  MoveL 1169 to (549.24, 512.97, 16) mm, rotated rx -180 ry 0 rz 160 deg; joints [7.081, 85.862, -31.558, -147.805, 58.7, 161.888]
  Set speed (17.5 mm/s)
  Call Extruder(1124.88314)
  MoveL 1170 to (548.96, 514.02, 16) mm, rotated rx -180 ry 0 rz 160 deg; joints [7.204, 85.828, -31.485, -147.681, 58.771, 161.841]
  Set speed (17.5 mm/s)
  Call Extruder(1131.34964)
  MoveL 1171 to (548.37, 515.94, 16) mm, rotated rx -180 ry 0 rz 160 deg; joints [7.43, 85.752, -31.322, -147.46, 58.916, 161.767]
  Set speed (17.5 mm/s)
  Call Extruder(1135.34697)
  MoveL 1172 to (547.97, 517.11, 16) mm, rotated rx 180 ry 0 rz 160 deg; joints [7.568, 85.697, -31.202, -147.327, 59.013, 161.728]
  Set speed (17.5 mm/s)
  Call Extruder(1138.01654)
  MoveL 1173 to (547.69, 517.88, 16) mm, rotated rx -180 ry 0 rz 160 deg; joints [7.66, 85.658, -31.119, -147.24, 59.08, 161.704]
  Set speed (17.5 mm/s)
  Call Extruder(1141.53682)
  MoveL 1174 to (547.29, 518.9, 16) mm, rotated rx -180 ry 0 rz 160 deg; joints [7.781, 85.601, -30.995, -147.127, 59.174, 161.677]
  Set speed (17.5 mm/s)
  Call Extruder(1144.91482)
  MoveL 1175 to (546.9, 519.87, 16) mm, rotated rx 180 ry 0 rz 160 deg; joints [7.897, 85.544, -30.872, -147.021, 59.266, 161.653]
  Set speed (17.5 mm/s)
  Call Extruder(1151.46736)
  MoveL 1176 to (546.07, 521.72, 16) mm, rotated rx -180 ry 0 rz 160 deg; joints [8.12, 85.42, -30.605, -146.821, 59.456, 161.619]
  Call Extruder(1154.81875)
  MoveL 1177 to (545.61, 522.65, 16) mm, rotated rx 180 ry 0 rz 160 deg; joints [8.233, 85.352, -30.456, -146.722, 59.559, 161.607]
  Set speed (17.5 mm/s)
  Call Extruder(1158.37572)
  MoveL 1178 to (545.12, 523.64, 16) mm, rotated rx -180 ry 0 rz 160 deg; joints [8.353, 85.275, -30.29, -146.619, 59.671, 161.597]
  Call Extruder(1161.73090)
  MoveL 1179 to (544.62, 524.55, 16) mm, rotated rx 180 ry 0 rz 160 deg; joints [8.465, 85.198, -30.123, -146.525, 59.782, 161.592]
  Set speed (17.5 mm/s)
  Call Extruder(1165.06713)
  MoveL 1180 to (544.12, 525.45, 16) mm, rotated rx -180 ry 0 rz 160 deg; joints [8.576, 85.119, -29.952, -146.433, 59.894, 161.59]
  Set speed (17.5 mm/s)
  Call Extruder(1169.60064)
  MoveL 1181 to (543.4, 526.66, 16) mm, rotated rx 180 ry 0 rz 160 deg; joints [8.726, 85.006, -29.706, -146.311, 60.051, 161.593]
  Set speed (17.5 mm/s)
  Call Extruder(1175.11317)
  MoveL 1182 to (542.48, 528.1, 16) mm, rotated rx 180 ry 0 rz 160 deg; joints [8.905, 84.859, -29.387, -146.17, 60.251, 161.605]
  Set speed (17.5 mm/s)
  Call Extruder(1178.53672)
  MoveL 1183 to (541.88, 528.97, 16) mm, rotated rx -180 ry 0 rz 160 deg; joints [9.016, 84.764, -29.18, -146.085, 60.379, 161.618]
  Set speed (17.5 mm/s)
  Call Extruder(1181.80346)
  MoveL 1184 to (541.3, 529.8, 16) mm, rotated rx 180 ry 0 rz 160 deg; joints [9.12, 84.67, -28.975, -146.005, 60.504, 161.632]
  Call Extruder(1185.22640)
  MoveL 1185 to (540.67, 530.65, 16) mm, rotated rx 180 ry 0 rz 160 deg; joints [9.229, 84.568, -28.753, -145.925, 60.638, 161.651]
  Set speed (17.5 mm/s)
  Call Extruder(1188.52738)
  MoveL 1186 to (540.05, 531.47, 16) mm, rotated rx -180 ry 0 rz 160 deg; joints [9.333, 84.467, -28.534, -145.849, 60.769, 161.672]
  Call Extruder(1191.91987)
  MoveL 1187 to (539.39, 532.28, 16) mm, rotated rx 180 ry 0 rz 160 deg; joints [9.439, 84.361, -28.3, -145.774, 60.907, 161.698]
  Set speed (17.5 mm/s)
  Call Extruder(1195.33158)
  MoveL 1188 to (538.71, 533.09, 16) mm, rotated rx 180 ry 0 rz 160 deg; joints [9.544, 84.25, -28.058, -145.7, 61.049, 161.727]
  Set speed (17.5 mm/s)
  Call Extruder(1198.69325)
  MoveL 1189 to (538.03, 533.88, 16) mm, rotated rx 180 ry 0 rz 160 deg; joints [9.647, 84.139, -27.814, -145.63, 61.19, 161.758]
  Set speed (17.5 mm/s)
  Call Extruder(1202.01515)
  MoveL 1190 to (537.33, 534.64, 16) mm, rotated rx 180 ry 0 rz 160 deg; joints [9.748, 84.026, -27.567, -145.563, 61.333, 161.792]
  Set speed (17.5 mm/s)
  Call Extruder(1205.37905)
  MoveL 1191 to (536.62, 535.4, 16) mm, rotated rx -180 ry 0 rz 160 deg; joints [9.849, 83.909, -27.31, -145.497, 61.479, 161.83]
  Call Extruder(1208.76243)
  MoveL 1192 to (535.88, 536.14, 16) mm, rotated rx -180 ry 0 rz 160 deg; joints [9.949, 83.789, -27.047, -145.432, 61.629, 161.871]
  Call Extruder(1212.12100)
  MoveL 1193 to (535.14, 536.87, 16) mm, rotated rx 180 ry 0 rz 160 deg; joints [10.047, 83.667, -26.779, -145.371, 61.779, 161.915]
  Call Extruder(1215.53799)
  MoveL 1194 to (534.36, 537.59, 16) mm, rotated rx -180 ry 0 rz 160 deg; joints [10.146, 83.541, -26.502, -145.311, 61.934, 161.962]
  Set speed (17.5 mm/s)
  Call Extruder(1218.83854)
  MoveL 1195 to (533.6, 538.27, 16) mm, rotated rx -180 ry 0 rz 160 deg; joints [10.24, 83.417, -26.228, -145.255, 62.087, 162.011]
  Set speed (17.5 mm/s)
  Call Extruder(1222.23079)
  MoveL 1196 to (532.8, 538.96, 16) mm, rotated rx 180 ry 0 rz 160 deg; joints [10.335, 83.287, -25.941, -145.199, 62.245, 162.065]
  Set speed (17.5 mm/s)
  Call Extruder(1225.64774)
  MoveL 1197 to (531.99, 539.63, 16) mm, rotated rx 180 ry 0 rz 160 deg; joints [10.43, 83.154, -25.648, -145.146, 62.406, 162.121]
  Set speed (17.5 mm/s)
  Call Extruder(1228.34274)
  MoveL 1198 to (531.33, 540.15, 16) mm, rotated rx 180 ry 0 rz 160 deg; joints [10.504, 83.048, -25.413, -145.105, 62.534, 162.167]
  Set speed (17.5 mm/s)
  Call Extruder(1232.24907)
  MoveL 1199 to (530.37, 540.88, 16) mm, rotated rx 180 ry 0 rz 160 deg; joints [10.609, 82.892, -25.067, -145.048, 62.722, 162.238]
  Set speed (17.5 mm/s)
  Call Extruder(1235.63039)
  MoveL 1200 to (529.52, 541.5, 16) mm, rotated rx 180 ry 0 rz 160 deg; joints [10.698, 82.755, -24.763, -145.002, 62.886, 162.302]
  Set speed (17.5 mm/s)
  Call Extruder(1238.99206)
  MoveL 1201 to (528.67, 542.1, 16) mm, rotated rx 180 ry 0 rz 160 deg; joints [10.786, 82.617, -24.456, -144.958, 63.051, 162.368]
  Call Extruder(1242.35571)
  MoveL 1202 to (527.8, 542.67, 16) mm, rotated rx -180 ry 0 rz 160 deg; joints [10.872, 82.477, -24.145, -144.916, 63.217, 162.437]
  Set speed (17.5 mm/s)
  Call Extruder(1245.76604)
  MoveL 1203 to (526.91, 543.24, 16) mm, rotated rx -180 ry 0 rz 160 deg; joints [10.958, 82.333, -23.825, -144.875, 63.387, 162.509]
  Set speed (17.5 mm/s)
  Call Extruder(1249.75916)
  MoveL 1204 to (525.85, 543.88, 16) mm, rotated rx 180 ry 0 rz 160 deg; joints [11.056, 82.164, -23.447, -144.83, 63.587, 162.597]
  Set speed (17.5 mm/s)
  Call Extruder(1255.55529)
  MoveL 1205 to (524.29, 544.77, 16) mm, rotated rx 180 ry 0 rz 160 deg; joints [11.195, 81.914, -22.888, -144.771, 63.881, 162.73]
  Set speed (17.5 mm/s)
  Call Extruder(1258.01050)
  MoveL 1206 to (523.62, 545.13, 16) mm, rotated rx -180 ry 0 rz 160 deg; joints [11.252, 81.808, -22.649, -144.747, 64.006, 162.788]
  Set speed (17.5 mm/s)
  Call Extruder(1261.12140)
  MoveL 1207 to (522.76, 545.56, 16) mm, rotated rx 180 ry 0 rz 160 deg; joints [11.323, 81.671, -22.342, -144.719, 64.166, 162.865]
  Set speed (17.5 mm/s)
  Call Extruder(1265.86908)
  MoveL 1208 to (521.44, 546.2, 16) mm, rotated rx 180 ry 0 rz 160 deg; joints [11.428, 81.461, -21.869, -144.681, 64.411, 162.984]
  Set speed (17.5 mm/s)
  Call Extruder(1269.35473)
  MoveL 1209 to (520.45, 546.64, 16) mm, rotated rx 180 ry 0 rz 160 deg; joints [11.503, 81.305, -21.519, -144.655, 64.592, 163.075]
  Call Extruder(1272.87309)
  MoveL 1210 to (519.45, 547.07, 16) mm, rotated rx 180 ry 0 rz 160 deg; joints [11.578, 81.148, -21.164, -144.63, 64.775, 163.168]
  Set speed (17.5 mm/s)
  Call Extruder(1279.51361)
  MoveL 1211 to (517.54, 547.82, 16) mm, rotated rx 180 ry 0 rz 160 deg; joints [11.712, 80.848, -20.484, -144.591, 65.123, 163.351]
  Set speed (17.5 mm/s)
  Call Extruder(1286.22822)
  MoveL 1212 to (515.57, 548.49, 16) mm, rotated rx 180 ry 0 rz 160 deg; joints [11.84, 80.542, -19.789, -144.56, 65.477, 163.543]
  Set speed (17.4 mm/s)
  Call Extruder(1290.32257)
  MoveL 1213 to (514.36, 548.86, 16) mm, rotated rx -180 ry 0 rz 160 deg; joints [11.914, 80.354, -19.361, -144.545, 65.693, 163.663]
  Set speed (17.5 mm/s)
  Call Extruder(1292.76941)
  MoveL 1214 to (513.63, 549.07, 16) mm, rotated rx -180 ry 0 rz 160 deg; joints [11.957, 80.242, -19.105, -144.538, 65.823, 163.736]
  Set speed (17.5 mm/s)
  Call Extruder(1295.71612)
  MoveL 1215 to (512.75, 549.3, 16) mm, rotated rx 180 ry 0 rz 160 deg; joints [12.006, 80.106, -18.794, -144.531, 65.979, 163.826]
  Set speed (17.5 mm/s)
  Call Extruder(1299.58645)
  MoveL 1216 to (511.59, 549.59, 16) mm, rotated rx 180 ry 0 rz 160 deg; joints [12.07, 79.928, -18.386, -144.523, 66.184, 163.945]
  Set speed (17.5 mm/s)
  Call Extruder(1306.36625)
  MoveL 1217 to (509.53, 550.03, 16) mm, rotated rx -180 ry 0 rz 160 deg; joints [12.175, 79.615, -17.666, -144.516, 66.544, 164.159]
  Set speed (17.5 mm/s)
  Call Extruder(1313.14810)
  MoveL 1218 to (507.46, 550.38, 16) mm, rotated rx 180 ry 0 rz 160 deg; joints [12.27, 79.301, -16.941, -144.519, 66.905, 164.379]
  Set speed (17.5 mm/s)
  Call Extruder(1319.69345)
  MoveL 1219 to (505.45, 550.64, 16) mm, rotated rx 180 ry 0 rz 160 deg; joints [12.354, 78.998, -16.239, -144.53, 67.252, 164.596]
  Set speed (17.5 mm/s)
  Call Extruder(1326.55936)
  MoveL 1220 to (503.33, 550.82, 16) mm, rotated rx -180 ry 0 rz 160 deg; joints [12.432, 78.681, -15.501, -144.549, 67.615, 164.829]
  Set speed (17.5 mm/s)
  Call Extruder(1333.32860)
  MoveL 1221 to (501.24, 550.91, 16) mm, rotated rx 180 ry 0 rz 160 deg; joints [12.499, 78.369, -14.774, -144.578, 67.972, 165.063]
  Set speed (17.5 mm/s)
  Call Extruder(1339.97617)
  MoveL 1222 to (499.18, 550.92, 16) mm, rotated rx -180 ry 0 rz 160 deg; joints [12.556, 78.066, -14.061, -144.614, 68.32, 165.297]
  Set speed (10.0 mm/s)
  MoveL 1223 to (499.18, 550.92, 20) mm, rotated rx 180 ry 0 rz 160 deg; joints [12.556, 77.328, -13.499, -144.573, 68.176, 165.187]
  Set speed (120.0 mm/s)
  MoveL 1224 to (499.16, 551.9, 20) mm, rotated rx 180 ry 0 rz 160 deg; joints [12.676, 77.358, -13.57, -144.439, 68.174, 165.115]
  Set speed (17.5 mm/s)
  Call Extruder(1346.89767)
  MoveL 1225 to (497.02, 551.82, 20) mm, rotated rx 180 ry 0 rz 160 deg; joints [12.725, 77.043, -12.831, -144.486, 68.531, 165.362]
  Set speed (17.5 mm/s)
  Call Extruder(1353.77145)
  MoveL 1226 to (494.9, 551.66, 20) mm, rotated rx 180 ry 0 rz 160 deg; joints [12.763, 76.734, -12.101, -144.541, 68.883, 165.609]
  Call Extruder(1360.44876)
  MoveL 1227 to (492.84, 551.41, 20) mm, rotated rx 180 ry 0 rz 160 deg; joints [12.791, 76.436, -11.396, -144.603, 69.222, 165.852]
  Set speed (17.5 mm/s)
  Call Extruder(1367.36675)
  MoveL 1228 to (490.72, 551.07, 20) mm, rotated rx 180 ry 0 rz 160 deg; joints [12.808, 76.131, -10.67, -144.676, 69.57, 166.106]
  Set speed (17.5 mm/s)
  Call Extruder(1374.35141)
  MoveL 1229 to (488.6, 550.64, 20) mm, rotated rx -180 ry 0 rz 160 deg; joints [12.814, 75.828, -9.943, -144.76, 69.917, 166.364]
  Set speed (17.5 mm/s)
  Call Extruder(1381.22915)
  MoveL 1230 to (486.53, 550.13, 20) mm, rotated rx 180 ry 0 rz 160 deg; joints [12.81, 75.533, -9.236, -144.851, 70.253, 166.619]
  Call Extruder(1387.89760)
  MoveL 1231 to (484.55, 549.56, 20) mm, rotated rx 180 ry 0 rz 160 deg; joints [12.794, 75.252, -8.558, -144.948, 70.575, 166.867]
  Set speed (17.5 mm/s)
  Call Extruder(1394.66926)
  MoveL 1232 to (482.56, 548.89, 20) mm, rotated rx 180 ry 0 rz 160 deg; joints [12.767, 74.972, -7.877, -145.057, 70.896, 167.119]
  Set speed (17.5 mm/s)
  Call Extruder(1398.28337)
  MoveL 1233 to (481.51, 548.5, 20) mm, rotated rx 180 ry 0 rz 160 deg; joints [12.747, 74.825, -7.518, -145.118, 71.065, 167.254]
  Call Extruder(1401.87388)
  MoveL 1234 to (480.48, 548.1, 20) mm, rotated rx -180 ry 0 rz 160 deg; joints [12.726, 74.68, -7.164, -145.181, 71.232, 167.387]
  Set speed (17.5 mm/s)
  Call Extruder(1406.78546)
  MoveL 1235 to (479.08, 547.51, 20) mm, rotated rx 180 ry 0 rz 160 deg; joints [12.691, 74.484, -6.685, -145.272, 71.458, 167.569]
  Set speed (17.5 mm/s)
  Call Extruder(1411.85900)
  MoveL 1236 to (477.65, 546.85, 20) mm, rotated rx 180 ry 0 rz 160 deg; joints [12.649, 74.285, -6.196, -145.371, 71.687, 167.757]
  Set speed (17.5 mm/s)
  Call Extruder(1416.96547)
  MoveL 1237 to (476.23, 546.15, 20) mm, rotated rx -180 ry 0 rz 160 deg; joints [12.6, 74.088, -5.71, -145.475, 71.915, 167.945]
  Set speed (17.5 mm/s)
  Call Extruder(1422.63061)
  MoveL 1238 to (474.69, 545.32, 20) mm, rotated rx 180 ry 0 rz 160 deg; joints [12.537, 73.874, -5.18, -145.597, 72.163, 168.153]
  Set speed (17.5 mm/s)
  Call Extruder(1425.60662)
  MoveL 1239 to (473.89, 544.87, 20) mm, rotated rx 180 ry 0 rz 160 deg; joints [12.501, 73.763, -4.905, -145.664, 72.291, 168.262]
  Set speed (17.5 mm/s)
  Call Extruder(1429.03570)
  MoveL 1240 to (472.97, 544.32, 20) mm, rotated rx 180 ry 0 rz 160 deg; joints [12.457, 73.637, -4.591, -145.743, 72.437, 168.387]
  Call Extruder(1432.47238)
  MoveL 1241 to (472.07, 543.76, 20) mm, rotated rx -180 ry 0 rz 160 deg; joints [12.41, 73.513, -4.28, -145.825, 72.582, 168.512]
  Set speed (17.5 mm/s)
  Call Extruder(1435.86869)
  MoveL 1242 to (471.19, 543.18, 20) mm, rotated rx -180 ry 0 rz 160 deg; joints [12.36, 73.391, -3.976, -145.908, 72.723, 168.634]
  Set speed (17.5 mm/s)
  Call Extruder(1439.36515)
  MoveL 1243 to (470.29, 542.57, 20) mm, rotated rx -180 ry 0 rz 160 deg; joints [12.306, 73.268, -3.667, -145.996, 72.867, 168.759]
  Set speed (17.5 mm/s)
  Call Extruder(1442.74341)
  MoveL 1244 to (469.44, 541.96, 20) mm, rotated rx 180 ry 0 rz 160 deg; joints [12.251, 73.151, -3.372, -146.082, 73.003, 168.88]
  Set speed (17.5 mm/s)
  Call Extruder(1446.13527)
  MoveL 1245 to (468.6, 541.34, 20) mm, rotated rx 180 ry 0 rz 160 deg; joints [12.193, 73.035, -3.08, -146.172, 73.139, 169]
  Call Extruder(1449.64837)
  MoveL 1246 to (467.74, 540.67, 20) mm, rotated rx -180 ry 0 rz 160 deg; joints [12.129, 72.917, -2.782, -146.267, 73.276, 169.123]
  Set speed (17.5 mm/s)
  Call Extruder(1453.05307)
  MoveL 1247 to (466.92, 540, 20) mm, rotated rx 180 ry 0 rz 160 deg; joints [12.065, 72.805, -2.497, -146.362, 73.408, 169.242]
  Set speed (17.5 mm/s)
  Call Extruder(1456.40954)
  MoveL 1248 to (466.12, 539.33, 20) mm, rotated rx -180 ry 0 rz 160 deg; joints [11.999, 72.696, -2.22, -146.457, 73.536, 169.358]
  Set speed (17.5 mm/s)
  Call Extruder(1459.89153)
  MoveL 1249 to (465.31, 538.62, 20) mm, rotated rx 180 ry 0 rz 160 deg; joints [11.927, 72.585, -1.937, -146.558, 73.666, 169.478]
  Call Extruder(1463.26727)
  MoveL 1250 to (464.54, 537.91, 20) mm, rotated rx 180 ry 0 rz 160 deg; joints [11.855, 72.479, -1.667, -146.659, 73.79, 169.593]
  Set speed (17.5 mm/s)
  Call Extruder(1466.74547)
  MoveL 1251 to (463.76, 537.17, 20) mm, rotated rx -180 ry 0 rz 160 deg; joints [11.778, 72.372, -1.393, -146.764, 73.916, 169.71]
  Set speed (17.5 mm/s)
  Call Extruder(1470.14894)
  MoveL 1252 to (463.01, 536.42, 20) mm, rotated rx 180 ry 0 rz 160 deg; joints [11.7, 72.27, -1.13, -146.869, 74.036, 169.824]
  Set speed (17.5 mm/s)
  Call Extruder(1473.62936)
  MoveL 1253 to (462.26, 535.64, 20) mm, rotated rx -180 ry 0 rz 160 deg; joints [11.617, 72.167, -0.866, -146.98, 74.157, 169.939]
  Set speed (17.5 mm/s)
  Call Extruder(1476.95452)
  MoveL 1254 to (461.56, 534.89, 20) mm, rotated rx 180 ry 0 rz 160 deg; joints [11.535, 72.071, -0.618, -147.087, 74.27, 170.047]
  Set speed (17.5 mm/s)
  Call Extruder(1480.45766)
  MoveL 1255 to (460.84, 534.08, 20) mm, rotated rx -180 ry 0 rz 160 deg; joints [11.446, 71.972, -0.362, -147.202, 74.387, 170.161]
  Set speed (17.5 mm/s)
  Call Extruder(1483.42207)
  MoveL 1256 to (460.24, 533.38, 20) mm, rotated rx 180 ry 0 rz 160 deg; joints [11.368, 71.89, -0.149, -147.301, 74.483, 170.255]
  Set speed (17.5 mm/s)
  Call Extruder(1487.30579)
  MoveL 1257 to (459.48, 532.45, 20) mm, rotated rx 180 ry 0 rz 160 deg; joints [11.264, 71.785, 0.124, -147.433, 74.607, 170.378]
  Set speed (17.5 mm/s)
  Call Extruder(1490.73127)
  MoveL 1258 to (458.83, 531.62, 20) mm, rotated rx -180 ry 0 rz 160 deg; joints [11.168, 71.694, 0.359, -147.552, 74.713, 170.484]
  Set speed (17.5 mm/s)
  Call Extruder(1494.14375)
  MoveL 1259 to (458.19, 530.77, 20) mm, rotated rx -180 ry 0 rz 160 deg; joints [11.071, 71.606, 0.588, -147.672, 74.816, 170.589]
  Set speed (17.5 mm/s)
  Call Extruder(1497.58334)
  MoveL 1260 to (457.57, 529.9, 20) mm, rotated rx -180 ry 0 rz 160 deg; joints [10.97, 71.52, 0.814, -147.795, 74.918, 170.693]
  Set speed (17.5 mm/s)
  Call Extruder(1500.98572)
  MoveL 1261 to (456.97, 529.04, 20) mm, rotated rx 180 ry 0 rz 160 deg; joints [10.867, 71.437, 1.032, -147.919, 75.016, 170.794]
  Set speed (17.5 mm/s)
  Call Extruder(1504.45910)
  MoveL 1262 to (456.38, 528.14, 20) mm, rotated rx 180 ry 0 rz 160 deg; joints [10.761, 71.354, 1.25, -148.048, 75.113, 170.896]
  Set speed (17.5 mm/s)
  Call Extruder(1507.83348)
  MoveL 1263 to (455.82, 527.25, 20) mm, rotated rx -180 ry 0 rz 160 deg; joints [10.654, 71.276, 1.455, -148.174, 75.204, 170.994]
  Set speed (17.5 mm/s)
  Call Extruder(1511.23944)
  MoveL 1264 to (455.27, 526.35, 20) mm, rotated rx 180 ry 0 rz 160 deg; joints [10.545, 71.199, 1.657, -148.303, 75.294, 171.09]
  Call Extruder(1514.69572)
  MoveL 1265 to (454.74, 525.42, 20) mm, rotated rx -180 ry 0 rz 160 deg; joints [10.431, 71.124, 1.857, -148.436, 75.382, 171.187]
  Set speed (17.5 mm/s)
  Call Extruder(1517.51539)
  MoveL 1266 to (454.32, 524.66, 20) mm, rotated rx 180 ry 0 rz 160 deg; joints [10.337, 71.064, 2.015, -148.546, 75.451, 171.264]
  Set speed (17.5 mm/s)
  Call Extruder(1521.55599)
  MoveL 1267 to (453.74, 523.55, 20) mm, rotated rx 180 ry 0 rz 160 deg; joints [10.199, 70.981, 2.234, -148.706, 75.547, 171.373]
  Set speed (17.5 mm/s)
  Call Extruder(1524.99033)
  MoveL 1268 to (453.26, 522.59, 20) mm, rotated rx 180 ry 0 rz 160 deg; joints [10.079, 70.913, 2.415, -148.843, 75.626, 171.464]
  Set speed (17.5 mm/s)
  Call Extruder(1528.51455)
  MoveL 1269 to (452.8, 521.61, 20) mm, rotated rx 180 ry 0 rz 160 deg; joints [9.954, 70.846, 2.593, -148.985, 75.702, 171.555]
  Set speed (17.5 mm/s)
  Call Extruder(1531.83917)
  MoveL 1270 to (452.38, 520.67, 20) mm, rotated rx -180 ry 0 rz 160 deg; joints [9.834, 70.785, 2.757, -149.121, 75.773, 171.639]
  Set speed (17.5 mm/s)
  Call Extruder(1538.58210)
  MoveL 1271 to (451.59, 518.73, 20) mm, rotated rx -180 ry 0 rz 160 deg; joints [9.585, 70.668, 3.07, -149.401, 75.905, 171.805]
  Call Extruder(1545.63097)
  MoveL 1272 to (450.84, 516.68, 20) mm, rotated rx -180 ry 0 rz 160 deg; joints [9.316, 70.555, 3.373, -149.699, 76.031, 171.971]
  Call Extruder(1552.49327)
  MoveL 1273 to (450.2, 514.66, 20) mm, rotated rx 180 ry 0 rz 160 deg; joints [9.048, 70.455, 3.642, -149.994, 76.14, 172.124]
  Set speed (17.5 mm/s)
  Call Extruder(1559.18400)
  MoveL 1274 to (449.65, 512.65, 20) mm, rotated rx -180 ry 0 rz 160 deg; joints [8.779, 70.367, 3.88, -150.286, 76.234, 172.266]
  Set speed (17.5 mm/s)
  Call Extruder(1562.76659)
  MoveL 1275 to (449.4, 511.57, 20) mm, rotated rx 180 ry 0 rz 160 deg; joints [8.633, 70.324, 3.996, -150.443, 76.278, 172.339]
  Call Extruder(1566.05852)
  MoveL 1276 to (449.18, 510.58, 20) mm, rotated rx 180 ry 0 rz 160 deg; joints [8.498, 70.286, 4.098, -150.589, 76.316, 172.404]
  Set speed (17.5 mm/s)
  Call Extruder(1573.08116)
  MoveL 1277 to (448.78, 508.44, 20) mm, rotated rx -180 ry 0 rz 160 deg; joints [8.205, 70.214, 4.295, -150.903, 76.386, 172.537]
  Call Extruder(0.00000)
  Set speed (17.5 mm/s)
  Call Extruder(6.84930)
  MoveL 1278 to (448.48, 506.34, 20) mm, rotated rx -180 ry 0 rz 160 deg; joints [7.914, 70.153, 4.46, -151.212, 76.44, 172.659]
  Set speed (17.5 mm/s)
  Call Extruder(13.69641)
  MoveL 1279 to (448.26, 504.23, 20) mm, rotated rx 180 ry 0 rz 160 deg; joints [7.62, 70.102, 4.599, -151.522, 76.48, 172.772]
  Set speed (17.5 mm/s)
  Call Extruder(20.39008)
  MoveL 1280 to (448.13, 502.16, 20) mm, rotated rx -180 ry 0 rz 160 deg; joints [7.329, 70.062, 4.709, -151.827, 76.505, 172.876]
  Call Extruder(27.31483)
  MoveL 1281 to (448.09, 500.02, 20) mm, rotated rx 180 ry 0 rz 160 deg; joints [7.026, 70.03, 4.795, -152.143, 76.516, 172.974]
  Set speed (17.5 mm/s)
  Call Extruder(33.56591)
  MoveL 1282 to (448.13, 498.08, 20) mm, rotated rx 180 ry 0 rz 160 deg; joints [6.75, 70.01, 4.85, -152.428, 76.513, 173.056]
  Set speed (17.5 mm/s)
  Call Extruder(39.66263)
  MoveL 1283 to (448.23, 496.19, 20) mm, rotated rx -180 ry 0 rz 160 deg; joints [6.48, 69.998, 4.881, -152.706, 76.498, 173.13]
  Call Extruder(46.07765)
  MoveL 1284 to (448.41, 494.21, 20) mm, rotated rx 180 ry 0 rz 160 deg; joints [6.195, 69.995, 4.891, -152.997, 76.47, 173.201]
  Set speed (17.5 mm/s)
  Call Extruder(51.90887)
  MoveL 1285 to (448.65, 492.42, 20) mm, rotated rx 180 ry 0 rz 160 deg; joints [5.936, 69.999, 4.879, -153.261, 76.432, 173.26]
  Call Extruder(58.24782)
  MoveL 1286 to (448.97, 490.48, 20) mm, rotated rx -180 ry 0 rz 160 deg; joints [5.656, 70.012, 4.845, -153.545, 76.38, 173.317]
  Set speed (17.5 mm/s)
  Call Extruder(64.31632)
  MoveL 1287 to (449.35, 488.64, 20) mm, rotated rx 180 ry 0 rz 160 deg; joints [5.388, 70.032, 4.79, -153.815, 76.318, 173.366]
  Set speed (17.5 mm/s)
  Call Extruder(70.48045)
  MoveL 1288 to (449.8, 486.78, 20) mm, rotated rx -180 ry 0 rz 160 deg; joints [5.118, 70.06, 4.712, -154.086, 76.242, 173.409]
  Set speed (17.5 mm/s)
  Call Extruder(76.66227)
  MoveL 1289 to (450.32, 484.94, 20) mm, rotated rx 180 ry 0 rz 160 deg; joints [4.849, 70.097, 4.612, -154.354, 76.155, 173.446]
  Set speed (17.5 mm/s)
  Call Extruder(82.76319)
  MoveL 1290 to (450.9, 483.14, 20) mm, rotated rx -180 ry 0 rz 160 deg; joints [4.586, 70.141, 4.492, -154.615, 76.056, 173.477]
  Call Extruder(89.07136)
  MoveL 1291 to (451.57, 481.31, 20) mm, rotated rx -180 ry 0 rz 160 deg; joints [4.317, 70.195, 4.346, -154.881, 75.942, 173.503]
  Call Extruder(95.23992)
  MoveL 1292 to (452.29, 479.54, 20) mm, rotated rx -180 ry 0 rz 160 deg; joints [4.058, 70.255, 4.182, -155.135, 75.819, 173.523]
  Call Extruder(101.24751)
  MoveL 1293 to (453.06, 477.84, 20) mm, rotated rx 180 ry 0 rz 160 deg; joints [3.81, 70.322, 4.001, -155.377, 75.687, 173.536]
  Set speed (17.5 mm/s)
  Call Extruder(107.57777)
  MoveL 1294 to (453.93, 476.08, 20) mm, rotated rx -180 ry 0 rz 160 deg; joints [3.553, 70.4, 3.79, -155.627, 75.537, 173.544]
  Call Extruder(113.65141)
  MoveL 1295 to (454.83, 474.43, 20) mm, rotated rx 180 ry 0 rz 160 deg; joints [3.312, 70.483, 3.567, -155.86, 75.382, 173.547]
  Set speed (17.5 mm/s)
  Call Extruder(119.90561)
  MoveL 1296 to (455.81, 472.76, 20) mm, rotated rx 180 ry 0 rz 160 deg; joints [3.068, 70.576, 3.315, -156.093, 75.21, 173.544]
  Set speed (17.5 mm/s)
  Call Extruder(125.99893)
  MoveL 1297 to (456.83, 471.17, 20) mm, rotated rx -180 ry 0 rz 160 deg; joints [2.837, 70.675, 3.051, -156.313, 75.033, 173.536]
  Set speed (17.5 mm/s)
  Call Extruder(132.15800)
  MoveL 1298 to (457.92, 469.6, 20) mm, rotated rx -180 ry 0 rz 160 deg; joints [2.609, 70.782, 2.764, -156.528, 74.843, 173.522]
  Call Extruder(138.31119)
  MoveL 1299 to (459.07, 468.07, 20) mm, rotated rx 180 ry 0 rz 160 deg; joints [2.388, 70.897, 2.458, -156.735, 74.642, 173.504]
  Set speed (17.5 mm/s)
  Call Extruder(144.56702)
  MoveL 1300 to (460.29, 466.57, 20) mm, rotated rx 180 ry 0 rz 160 deg; joints [2.171, 71.022, 2.127, -156.937, 74.428, 173.479]
  Set speed (17.5 mm/s)
  Call Extruder(150.65295)
  MoveL 1301 to (461.53, 465.15, 20) mm, rotated rx -180 ry 0 rz 160 deg; joints [1.966, 71.15, 1.787, -157.124, 74.209, 173.45]
  Set speed (17.5 mm/s)
  Call Extruder(156.90741)
  MoveL 1302 to (462.86, 463.74, 20) mm, rotated rx 180 ry 0 rz 160 deg; joints [1.764, 71.29, 1.418, -157.308, 73.975, 173.416]
  Call Extruder(162.86927)
  MoveL 1303 to (464.17, 462.44, 20) mm, rotated rx -180 ry 0 rz 160 deg; joints [1.579, 71.43, 1.05, -157.475, 73.743, 173.378]
  Call Extruder(169.18566)
  MoveL 1304 to (465.61, 461.11, 20) mm, rotated rx 180 ry 0 rz 160 deg; joints [1.39, 71.586, 0.642, -157.641, 73.488, 173.332]
  Set speed (17.5 mm/s)
  Call Extruder(175.35316)
  MoveL 1305 to (467.07, 459.87, 20) mm, rotated rx 180 ry 0 rz 160 deg; joints [1.215, 71.745, 0.226, -157.794, 73.231, 173.283]
  Set speed (17.5 mm/s)
  Call Extruder(181.85609)
  MoveL 1306 to (468.65, 458.63, 20) mm, rotated rx -180 ry 0 rz 160 deg; joints [1.039, 71.921, -0.23, -157.944, 72.95, 173.225]
  Set speed (17.5 mm/s)
  Call Extruder(187.18333)
  MoveL 1307 to (469.98, 457.65, 20) mm, rotated rx 180 ry 0 rz 160 deg; joints [0.903, 72.071, -0.617, -158.058, 72.714, 173.174]
  Set speed (17.5 mm/s)
  Call Extruder(193.82493)
  MoveL 1308 to (471.68, 456.49, 20) mm, rotated rx -180 ry 0 rz 160 deg; joints [0.742, 72.264, -1.116, -158.19, 72.412, 173.105]
  Set speed (17.5 mm/s)
  Call Extruder(200.07187)
  MoveL 1309 to (473.32, 455.47, 20) mm, rotated rx 180 ry 0 rz 160 deg; joints [0.6, 72.454, -1.602, -158.303, 72.119, 173.035]
  Call Extruder(206.24160)
  MoveL 1310 to (474.98, 454.52, 20) mm, rotated rx -180 ry 0 rz 160 deg; joints [0.469, 72.648, -2.097, -158.403, 71.824, 172.96]
  Set speed (17.5 mm/s)
  Call Extruder(212.42019)
  MoveL 1311 to (476.67, 453.63, 20) mm, rotated rx 180 ry 0 rz 160 deg; joints [0.348, 72.848, -2.606, -158.493, 71.521, 172.881]
  Set speed (17.5 mm/s)
  Call Extruder(218.39493)
  MoveL 1312 to (478.34, 452.83, 20) mm, rotated rx -180 ry 0 rz 160 deg; joints [0.239, 73.048, -3.112, -158.569, 71.223, 172.799]
  Call Extruder(224.75574)
  MoveL 1313 to (480.15, 452.04, 20) mm, rotated rx 180 ry 0 rz 160 deg; joints [0.133, 73.267, -3.664, -158.639, 70.9, 172.707]
  Set speed (17.5 mm/s)
  Call Extruder(230.75775)
  MoveL 1314 to (481.88, 451.36, 20) mm, rotated rx 180 ry 0 rz 160 deg; joints [0.041, 73.48, -4.197, -158.694, 70.59, 172.615]
  Set speed (17.5 mm/s)
  Call Extruder(237.09101)
  MoveL 1315 to (483.73, 450.71, 20) mm, rotated rx 180 ry 0 rz 160 deg; joints [-0.045, 73.71, -4.771, -158.74, 70.258, 172.513]
  Set speed (17.5 mm/s)
  Call Extruder(243.20984)
  MoveL 1316 to (485.54, 450.14, 20) mm, rotated rx 180 ry 0 rz 160 deg; joints [-0.118, 73.937, -5.337, -158.773, 69.933, 172.409]
  Set speed (17.5 mm/s)
  Call Extruder(249.37088)
  MoveL 1317 to (487.39, 449.65, 20) mm, rotated rx -180 ry 0 rz 160 deg; joints [-0.183, 74.172, -5.918, -158.796, 69.602, 172.299]
  Call Extruder(255.54669)
  MoveL 1318 to (489.25, 449.21, 20) mm, rotated rx -180 ry 0 rz 160 deg; joints [-0.239, 74.413, -6.51, -158.807, 69.266, 172.184]
  Set speed (17.5 mm/s)
  Call Extruder(261.60188)
  MoveL 1319 to (491.09, 448.86, 20) mm, rotated rx 180 ry 0 rz 160 deg; joints [-0.284, 74.653, -7.1, -158.807, 68.934, 172.066]
  Set speed (17.5 mm/s)
  Call Extruder(267.49098)
  MoveL 1320 to (492.89, 448.58, 20) mm, rotated rx -180 ry 0 rz 160 deg; joints [-0.32, 74.891, -7.681, -158.796, 68.609, 171.946]
  Call Extruder(273.99527)
  MoveL 1321 to (494.9, 448.34, 20) mm, rotated rx -180 ry 0 rz 160 deg; joints [-0.348, 75.159, -8.332, -158.772, 68.248, 171.808]
  Set speed (17.5 mm/s)
  Call Extruder(280.16768)
  MoveL 1322 to (496.8, 448.19, 20) mm, rotated rx -180 ry 0 rz 160 deg; joints [-0.367, 75.418, -8.957, -158.738, 67.904, 171.672]
  Call Extruder(286.42584)
  MoveL 1323 to (498.74, 448.11, 20) mm, rotated rx 180 ry 0 rz 160 deg; joints [-0.376, 75.684, -9.598, -158.692, 67.553, 171.529]
  Set speed (17.5 mm/s)
  Call Extruder(292.51904)
  MoveL 1324 to (500.63, 448.09, 20) mm, rotated rx 180 ry 0 rz 160 deg; joints [-0.376, 75.947, -10.229, -158.636, 67.211, 171.384]
  Set speed (17.5 mm/s)
  Call Extruder(298.76296)
  MoveL 1325 to (502.56, 448.15, 20) mm, rotated rx -180 ry 0 rz 160 deg; joints [-0.367, 76.219, -10.88, -158.568, 66.859, 171.23]
  Set speed (17.5 mm/s)
  Call Extruder(304.84597)
  MoveL 1326 to (504.44, 448.28, 20) mm, rotated rx -180 ry 0 rz 160 deg; joints [-0.349, 76.488, -11.52, -158.49, 66.517, 171.075]
  Set speed (17.5 mm/s)
  Call Extruder(310.88075)
  MoveL 1327 to (506.3, 448.48, 20) mm, rotated rx -180 ry 0 rz 160 deg; joints [-0.323, 76.758, -12.158, -158.403, 66.179, 170.916]
  Set speed (17.5 mm/s)
  Call Extruder(317.20333)
  MoveL 1328 to (508.24, 448.75, 20) mm, rotated rx -180 ry 0 rz 160 deg; joints [-0.287, 77.042, -12.829, -158.301, 65.825, 170.744]
  Set speed (17.5 mm/s)
  Call Extruder(323.33518)
  MoveL 1329 to (510.11, 449.08, 20) mm, rotated rx 180 ry 0 rz 160 deg; joints [-0.244, 77.321, -13.483, -158.192, 65.483, 170.572]
  Set speed (17.5 mm/s)
  Call Extruder(328.91158)
  MoveL 1330 to (511.8, 449.45, 20) mm, rotated rx 180 ry 0 rz 160 deg; joints [-0.198, 77.575, -14.079, -158.083, 65.174, 170.412]
  Call Extruder(335.60217)
  MoveL 1331 to (513.81, 449.96, 20) mm, rotated rx 180 ry 0 rz 160 deg; joints [-0.134, 77.882, -14.794, -157.942, 64.806, 170.213]
  Set speed (17.5 mm/s)
  Call Extruder(341.84087)
  MoveL 1332 to (515.67, 450.51, 20) mm, rotated rx 180 ry 0 rz 160 deg; joints [-0.066, 78.17, -15.462, -157.8, 64.466, 170.023]
  Set speed (17.5 mm/s)
  Call Extruder(348.08429)
  MoveL 1333 to (517.5, 451.13, 20) mm, rotated rx -180 ry 0 rz 160 deg; joints [0.011, 78.459, -16.129, -157.647, 64.129, 169.827]
  Call Extruder(354.17423)
  MoveL 1334 to (519.27, 451.8, 20) mm, rotated rx -180 ry 0 rz 160 deg; joints [0.092, 78.741, -16.779, -157.489, 63.803, 169.632]
  Call Extruder(360.41686)
  MoveL 1335 to (521.05, 452.55, 20) mm, rotated rx -180 ry 0 rz 160 deg; joints [0.183, 79.03, -17.443, -157.318, 63.474, 169.427]
  Call Extruder(366.58690)
  MoveL 1336 to (522.78, 453.36, 20) mm, rotated rx -180 ry 0 rz 160 deg; joints [0.281, 79.315, -18.095, -157.139, 63.153, 169.22]
  Set speed (17.5 mm/s)
  Call Extruder(372.59726)
  MoveL 1337 to (524.44, 454.21, 20) mm, rotated rx 180 ry 0 rz 160 deg; joints [0.382, 79.592, -18.726, -156.957, 62.847, 169.014]
  Call Extruder(378.91663)
  MoveL 1338 to (526.15, 455.16, 20) mm, rotated rx -180 ry 0 rz 160 deg; joints [0.496, 79.882, -19.385, -156.757, 62.529, 168.793]
  Set speed (17.5 mm/s)
  Call Extruder(384.99300)
  MoveL 1339 to (527.76, 456.14, 20) mm, rotated rx -180 ry 0 rz 160 deg; joints [0.612, 80.159, -20.013, -156.556, 62.23, 168.577]
  Set speed (17.5 mm/s)
  Call Extruder(391.25117)
  MoveL 1340 to (529.38, 457.21, 20) mm, rotated rx 180 ry 0 rz 160 deg; joints [0.738, 80.442, -20.652, -156.341, 61.929, 168.351]
  Set speed (17.5 mm/s)
  Call Extruder(397.19940)
  MoveL 1341 to (530.88, 458.27, 20) mm, rotated rx 180 ry 0 rz 160 deg; joints [0.863, 80.709, -21.252, -156.13, 61.649, 168.133]
  Set speed (17.5 mm/s)
  Call Extruder(403.53259)
  MoveL 1342 to (532.44, 459.47, 20) mm, rotated rx -180 ry 0 rz 160 deg; joints [1.003, 80.99, -21.882, -155.897, 61.36, 167.897]
  Call Extruder(409.53413)
  MoveL 1343 to (533.87, 460.66, 20) mm, rotated rx -180 ry 0 rz 160 deg; joints [1.14, 81.253, -22.469, -155.67, 61.092, 167.671]
  Call Extruder(415.76527)
  MoveL 1344 to (535.31, 461.95, 20) mm, rotated rx -180 ry 0 rz 160 deg; joints [1.289, 81.521, -23.068, -155.428, 60.824, 167.434]
  Call Extruder(422.07973)
  MoveL 1345 to (536.72, 463.3, 20) mm, rotated rx -180 ry 0 rz 160 deg; joints [1.445, 81.789, -23.664, -155.177, 60.56, 167.191]
  Call Extruder(425.35628)
  MoveL 1346 to (537.43, 464.03, 20) mm, rotated rx 180 ry 0 rz 160 deg; joints [1.528, 81.926, -23.968, -155.044, 60.428, 167.065]
  Set speed (17.5 mm/s)
  Call Extruder(428.77503)
  MoveL 1347 to (538.15, 464.8, 20) mm, rotated rx 180 ry 0 rz 160 deg; joints [1.617, 82.067, -24.28, -154.903, 60.292, 166.932]
  Set speed (17.5 mm/s)
  Call Extruder(432.19134)
  MoveL 1348 to (538.86, 465.59, 20) mm, rotated rx -180 ry 0 rz 160 deg; joints [1.707, 82.206, -24.589, -154.761, 60.159, 166.799]
  Set speed (17.5 mm/s)
  Call Extruder(435.63311)
  MoveL 1349 to (539.56, 466.39, 20) mm, rotated rx -180 ry 0 rz 160 deg; joints [1.799, 82.345, -24.895, -154.617, 60.029, 166.665]
  Set speed (17.5 mm/s)
  Call Extruder(439.17845)
  MoveL 1350 to (540.27, 467.24, 20) mm, rotated rx -180 ry 0 rz 160 deg; joints [1.895, 82.486, -25.205, -154.467, 59.898, 166.527]
  Set speed (17.5 mm/s)
  Call Extruder(442.52401)
  MoveL 1351 to (540.91, 468.05, 20) mm, rotated rx -180 ry 0 rz 160 deg; joints [1.987, 82.617, -25.494, -154.323, 59.777, 166.396]
  Set speed (17.5 mm/s)
  Call Extruder(445.90952)
  MoveL 1352 to (541.55, 468.88, 20) mm, rotated rx -180 ry 0 rz 160 deg; joints [2.082, 82.747, -25.781, -154.177, 59.659, 166.264]
  Set speed (17.5 mm/s)
  Call Extruder(448.86173)
  MoveL 1353 to (542.09, 469.62, 20) mm, rotated rx 180 ry 0 rz 160 deg; joints [2.165, 82.859, -26.028, -154.049, 59.557, 166.148]
  Call Extruder(452.72753)
  MoveL 1354 to (542.78, 470.6, 20) mm, rotated rx 180 ry 0 rz 160 deg; joints [2.276, 83.003, -26.343, -153.88, 59.43, 165.997]
  Set speed (17.5 mm/s)
  Call Extruder(455.75332)
  MoveL 1355 to (543.31, 471.38, 20) mm, rotated rx -180 ry 0 rz 160 deg; joints [2.364, 83.114, -26.587, -153.746, 59.332, 165.879]
  Call Extruder(459.59881)
  MoveL 1356 to (543.95, 472.38, 20) mm, rotated rx -180 ry 0 rz 160 deg; joints [2.477, 83.252, -26.889, -153.575, 59.213, 165.729]
  Set speed (17.5 mm/s)
  Call Extruder(463.01746)
  MoveL 1357 to (544.51, 473.28, 20) mm, rotated rx -180 ry 0 rz 160 deg; joints [2.579, 83.372, -27.151, -153.422, 59.111, 165.596]
  Set speed (17.5 mm/s)
  Call Extruder(466.46723)
  MoveL 1358 to (545.05, 474.21, 20) mm, rotated rx 180 ry 0 rz 160 deg; joints [2.683, 83.49, -27.41, -153.267, 59.011, 165.462]
  Set speed (17.5 mm/s)
  Call Extruder(471.90101)
  MoveL 1359 to (545.86, 475.68, 20) mm, rotated rx -180 ry 0 rz 160 deg; joints [2.848, 83.671, -27.805, -153.022, 58.862, 165.253]
  Set speed (17.5 mm/s)
  Call Extruder(476.86174)
  MoveL 1360 to (546.56, 477.05, 20) mm, rotated rx -180 ry 0 rz 160 deg; joints [3.002, 83.83, -28.15, -152.797, 58.735, 165.063]
  Set speed (17.5 mm/s)
  Call Extruder(482.73409)
  MoveL 1361 to (547.34, 478.69, 20) mm, rotated rx -180 ry 0 rz 160 deg; joints [3.186, 84.011, -28.545, -152.529, 58.594, 164.84]
  Set speed (17.5 mm/s)
  Call Extruder(490.40334)
  MoveL 1362 to (548.26, 480.88, 20) mm, rotated rx 180 ry 0 rz 160 deg; joints [3.432, 84.231, -29.022, -152.178, 58.43, 164.555]
  Set speed (17.5 mm/s)
  Call Extruder(497.19049)
  MoveL 1363 to (548.99, 482.85, 20) mm, rotated rx -180 ry 0 rz 160 deg; joints [3.653, 84.413, -29.416, -151.867, 58.303, 164.307]
  Set speed (17.5 mm/s)
  Call Extruder(500.81084)
  MoveL 1364 to (549.35, 483.91, 20) mm, rotated rx 180 ry 0 rz 160 deg; joints [3.772, 84.503, -29.612, -151.701, 58.242, 164.178]
  Set speed (17.5 mm/s)
  Call Extruder(504.13273)
  MoveL 1365 to (549.66, 484.89, 20) mm, rotated rx 180 ry 0 rz 160 deg; joints [3.881, 84.585, -29.789, -151.549, 58.188, 164.059]
  Set speed (17.5 mm/s)
  Call Extruder(511.08636)
  MoveL 1366 to (550.25, 486.97, 20) mm, rotated rx 180 ry 0 rz 160 deg; joints [4.113, 84.743, -30.13, -151.232, 58.091, 163.817]
  Call Extruder(517.86034)
  MoveL 1367 to (550.73, 489.01, 20) mm, rotated rx 180 ry 0 rz 160 deg; joints [4.342, 84.881, -30.429, -150.925, 58.015, 163.589]
  Call Extruder(524.78335)
  MoveL 1368 to (551.14, 491.11, 20) mm, rotated rx 180 ry 0 rz 160 deg; joints [4.578, 85.008, -30.701, -150.614, 57.955, 163.364]
  Call Extruder(531.56213)
  MoveL 1369 to (551.46, 493.19, 20) mm, rotated rx -180 ry 0 rz 160 deg; joints [4.811, 85.115, -30.932, -150.312, 57.914, 163.152]
  Set speed (17.5 mm/s)
  Call Extruder(538.57711)
  MoveL 1370 to (551.7, 495.35, 20) mm, rotated rx 180 ry 0 rz 160 deg; joints [5.054, 85.21, -31.137, -150.003, 57.89, 162.942]
  Set speed (17.5 mm/s)
  Call Extruder(545.33174)
  MoveL 1371 to (551.85, 497.44, 20) mm, rotated rx 180 ry 0 rz 160 deg; joints [5.29, 85.285, -31.297, -149.711, 57.886, 162.75]
  Set speed (17.5 mm/s)
  Call Extruder(552.17049)
  MoveL 1372 to (551.91, 499.56, 20) mm, rotated rx -180 ry 0 rz 160 deg; joints [5.529, 85.343, -31.423, -149.419, 57.899, 162.566]
  Set speed (17.5 mm/s)
  Call Extruder(559.11146)
  MoveL 1373 to (551.88, 501.71, 20) mm, rotated rx 180 ry 0 rz 160 deg; joints [5.773, 85.385, -31.513, -149.13, 57.931, 162.391]
  Set speed (17.5 mm/s)
  Call Extruder(565.86897)
  MoveL 1374 to (551.77, 503.8, 20) mm, rotated rx 180 ry 0 rz 160 deg; joints [6.011, 85.408, -31.562, -148.854, 57.981, 162.233]
  Call Extruder(572.64602)
  MoveL 1375 to (551.57, 505.89, 20) mm, rotated rx -180 ry 0 rz 160 deg; joints [6.25, 85.415, -31.576, -148.583, 58.048, 162.087]
  Set speed (17.5 mm/s)
  Call Extruder(579.67802)
  MoveL 1376 to (551.28, 508.05, 20) mm, rotated rx -180 ry 0 rz 160 deg; joints [6.498, 85.403, -31.551, -148.31, 58.136, 161.948]
  Set speed (17.5 mm/s)
  Call Extruder(586.42842)
  MoveL 1377 to (550.92, 510.11, 20) mm, rotated rx 180 ry 0 rz 160 deg; joints [6.735, 85.375, -31.49, -148.055, 58.237, 161.828]
  Set speed (17.5 mm/s)
  Call Extruder(593.33712)
  MoveL 1378 to (550.46, 512.21, 20) mm, rotated rx 180 ry 0 rz 160 deg; joints [6.978, 85.328, -31.39, -147.801, 58.358, 161.719]
  Set speed (17.5 mm/s)
  Call Extruder(596.73152)
  MoveL 1379 to (550.19, 513.22, 20) mm, rotated rx 180 ry 0 rz 160 deg; joints [7.096, 85.298, -31.325, -147.681, 58.425, 161.672]
  Set speed (17.5 mm/s)
  Call Extruder(600.32140)
  MoveL 1380 to (549.9, 514.3, 20) mm, rotated rx -180 ry 0 rz 160 deg; joints [7.222, 85.263, -31.251, -147.554, 58.498, 161.624]
  Set speed (17.5 mm/s)
  Call Extruder(606.81202)
  MoveL 1381 to (549.31, 516.22, 20) mm, rotated rx 180 ry 0 rz 160 deg; joints [7.448, 85.187, -31.086, -147.332, 58.644, 161.548]
  Call Extruder(613.77511)
  MoveL 1382 to (548.6, 518.26, 20) mm, rotated rx 180 ry 0 rz 160 deg; joints [7.689, 85.089, -30.876, -147.102, 58.815, 161.481]
  Set speed (17.5 mm/s)
  Call Extruder(620.57631)
  MoveL 1383 to (547.81, 520.21, 20) mm, rotated rx 180 ry 0 rz 160 deg; joints [7.922, 84.976, -30.633, -146.886, 58.998, 161.43]
  Set speed (17.5 mm/s)
  Call Extruder(624.13088)
  MoveL 1384 to (547.37, 521.22, 20) mm, rotated rx -180 ry 0 rz 160 deg; joints [8.043, 84.91, -30.491, -146.777, 59.1, 161.41]
  Set speed (17.5 mm/s)
  Call Extruder(627.38632)
  MoveL 1385 to (546.95, 522.14, 20) mm, rotated rx -180 ry 0 rz 160 deg; joints [8.153, 84.848, -30.357, -146.679, 59.196, 161.394]
  Set speed (17.5 mm/s)
  Call Extruder(630.88513)
  MoveL 1386 to (546.48, 523.11, 20) mm, rotated rx 180 ry 0 rz 160 deg; joints [8.271, 84.776, -30.202, -146.576, 59.303, 161.38]
  Set speed (17.5 mm/s)
  Call Extruder(634.33475)
  MoveL 1387 to (546, 524.07, 20) mm, rotated rx -180 ry 0 rz 160 deg; joints [8.387, 84.702, -30.042, -146.476, 59.412, 161.37]
  Set speed (17.5 mm/s)
  Call Extruder(637.83411)
  MoveL 1388 to (545.48, 525.02, 20) mm, rotated rx -180 ry 0 rz 160 deg; joints [8.504, 84.622, -29.87, -146.378, 59.526, 161.364]
  Set speed (17.5 mm/s)
  Call Extruder(641.18121)
  MoveL 1389 to (544.97, 525.93, 20) mm, rotated rx -180 ry 0 rz 160 deg; joints [8.615, 84.543, -29.697, -146.286, 59.639, 161.362]
  Set speed (17.5 mm/s)
  Call Extruder(645.47650)
  MoveL 1390 to (544.29, 527.07, 20) mm, rotated rx 180 ry 0 rz 160 deg; joints [8.757, 84.436, -29.466, -146.171, 59.787, 161.364]
  Set speed (17.5 mm/s)
  Call Extruder(648.04286)
  MoveL 1391 to (543.87, 527.75, 20) mm, rotated rx 180 ry 0 rz 160 deg; joints [8.841, 84.369, -29.32, -146.104, 59.879, 161.368]
  Set speed (17.5 mm/s)
  Call Extruder(651.48165)
  MoveL 1392 to (543.29, 528.64, 20) mm, rotated rx -180 ry 0 rz 160 deg; joints [8.953, 84.276, -29.12, -146.017, 60.004, 161.376]
  Set speed (17.5 mm/s)
  Call Extruder(654.87230)
  MoveL 1393 to (542.71, 529.51, 20) mm, rotated rx -180 ry 0 rz 160 deg; joints [9.062, 84.182, -28.916, -145.933, 60.13, 161.388]
  Call Extruder(658.36623)
  MoveL 1394 to (542.08, 530.4, 20) mm, rotated rx 180 ry 0 rz 160 deg; joints [9.174, 84.081, -28.697, -145.848, 60.264, 161.403]
  Set speed (17.5 mm/s)
  Call Extruder(661.88724)
  MoveL 1395 to (541.43, 531.27, 20) mm, rotated rx 180 ry 0 rz 160 deg; joints [9.286, 83.977, -28.47, -145.766, 60.401, 161.422]
  Set speed (17.5 mm/s)
  Call Extruder(665.17030)
  MoveL 1396 to (540.81, 532.08, 20) mm, rotated rx 180 ry 0 rz 160 deg; joints [9.389, 83.877, -28.252, -145.691, 60.531, 161.443]
  Set speed (17.5 mm/s)
  Call Extruder(668.59493)
  MoveL 1397 to (540.15, 532.91, 20) mm, rotated rx 180 ry 0 rz 160 deg; joints [9.496, 83.769, -28.017, -145.615, 60.67, 161.468]
  Set speed (17.5 mm/s)
  Call Extruder(672.08025)
  MoveL 1398 to (539.45, 533.74, 20) mm, rotated rx -180 ry 0 rz 160 deg; joints [9.604, 83.656, -27.771, -145.54, 60.814, 161.497]
  Set speed (17.5 mm/s)
  Call Extruder(675.49297)
  MoveL 1399 to (538.76, 534.53, 20) mm, rotated rx -180 ry 0 rz 160 deg; joints [9.708, 83.543, -27.525, -145.469, 60.957, 161.528]
  Call Extruder(678.85590)
  MoveL 1400 to (538.06, 535.3, 20) mm, rotated rx -180 ry 0 rz 160 deg; joints [9.81, 83.429, -27.275, -145.401, 61.101, 161.563]
  Set speed (17.5 mm/s)
  Call Extruder(682.37940)
  MoveL 1401 to (537.31, 536.1, 20) mm, rotated rx 180 ry 0 rz 160 deg; joints [9.915, 83.306, -27.008, -145.332, 61.253, 161.602]
  Set speed (17.5 mm/s)
  Call Extruder(685.79723)
  MoveL 1402 to (536.56, 536.85, 20) mm, rotated rx -180 ry 0 rz 160 deg; joints [10.016, 83.185, -26.742, -145.268, 61.404, 161.643]
  Set speed (17.5 mm/s)
  Call Extruder(689.14305)
  MoveL 1403 to (535.82, 537.57, 20) mm, rotated rx -180 ry 0 rz 160 deg; joints [10.114, 83.063, -26.476, -145.207, 61.553, 161.686]
  Set speed (17.5 mm/s)
  Call Extruder(695.21264)
  MoveL 1404 to (534.43, 538.85, 20) mm, rotated rx 180 ry 0 rz 160 deg; joints [10.288, 82.838, -25.982, -145.101, 61.829, 161.772]
  Set speed (17.5 mm/s)
  Call Extruder(699.40855)
  MoveL 1405 to (533.45, 539.7, 20) mm, rotated rx -180 ry 0 rz 160 deg; joints [10.406, 82.678, -25.63, -145.033, 62.023, 161.837]
  Set speed (17.5 mm/s)
  Call Extruder(702.90545)
  MoveL 1406 to (532.62, 540.39, 20) mm, rotated rx -180 ry 0 rz 160 deg; joints [10.503, 82.542, -25.331, -144.978, 62.187, 161.894]
  Set speed (17.5 mm/s)
  Call Extruder(706.26813)
  MoveL 1407 to (531.8, 541.03, 20) mm, rotated rx -180 ry 0 rz 160 deg; joints [10.595, 82.41, -25.039, -144.928, 62.346, 161.951]
  Set speed (17.5 mm/s)
  Call Extruder(709.70068)
  MoveL 1408 to (530.95, 541.67, 20) mm, rotated rx -180 ry 0 rz 160 deg; joints [10.688, 82.273, -24.735, -144.879, 62.511, 162.013]
  Set speed (17.5 mm/s)
  Call Extruder(713.15736)
  MoveL 1409 to (530.08, 542.31, 20) mm, rotated rx -180 ry 0 rz 160 deg; joints [10.779, 82.133, -24.426, -144.831, 62.677, 162.078]
  Set speed (17.5 mm/s)
  Call Extruder(716.56707)
  MoveL 1410 to (529.22, 542.91, 20) mm, rotated rx 180 ry 0 rz 160 deg; joints [10.868, 81.992, -24.115, -144.787, 62.844, 162.145]
  Set speed (17.5 mm/s)
  Call Extruder(720.01045)
  MoveL 1411 to (528.33, 543.5, 20) mm, rotated rx 180 ry 0 rz 160 deg; joints [10.956, 81.849, -23.798, -144.744, 63.013, 162.215]
  Set speed (17.5 mm/s)
  Call Extruder(723.39249)
  MoveL 1412 to (527.44, 544.06, 20) mm, rotated rx -180 ry 0 rz 160 deg; joints [11.041, 81.707, -23.482, -144.704, 63.181, 162.286]
  Set speed (17.5 mm/s)
  Call Extruder(726.96845)
  MoveL 1413 to (526.5, 544.64, 20) mm, rotated rx -180 ry 0 rz 160 deg; joints [11.13, 81.556, -23.145, -144.663, 63.359, 162.364]
  Set speed (17.5 mm/s)
  Call Extruder(730.28187)
  MoveL 1414 to (525.61, 545.16, 20) mm, rotated rx -180 ry 0 rz 160 deg; joints [11.21, 81.413, -22.828, -144.629, 63.526, 162.439]
  Set speed (17.5 mm/s)
  Call Extruder(733.10921)
  MoveL 1415 to (524.84, 545.58, 20) mm, rotated rx -180 ry 0 rz 160 deg; joints [11.277, 81.292, -22.556, -144.6, 63.668, 162.504]
  Set speed (17.5 mm/s)
  Call Extruder(739.07113)
  MoveL 1416 to (523.21, 546.44, 20) mm, rotated rx 180 ry 0 rz 160 deg; joints [11.414, 81.032, -21.975, -144.546, 63.971, 162.647]
  Set speed (17.5 mm/s)
  Call Extruder(743.92927)
  MoveL 1417 to (521.85, 547.09, 20) mm, rotated rx 180 ry 0 rz 160 deg; joints [11.522, 80.817, -21.494, -144.506, 64.22, 162.769]
  Call Extruder(747.49721)
  MoveL 1418 to (520.85, 547.54, 20) mm, rotated rx -180 ry 0 rz 160 deg; joints [11.599, 80.658, -21.137, -144.48, 64.404, 162.861]
  Set speed (17.5 mm/s)
  Call Extruder(750.90332)
  MoveL 1419 to (519.88, 547.96, 20) mm, rotated rx 180 ry 0 rz 160 deg; joints [11.671, 80.506, -20.795, -144.456, 64.58, 162.95]
  Set speed (17.5 mm/s)
  Call Extruder(757.79659)
  MoveL 1420 to (517.89, 548.73, 20) mm, rotated rx 180 ry 0 rz 160 deg; joints [11.811, 80.194, -20.092, -144.416, 64.939, 163.139]
  Set speed (17.5 mm/s)
  Call Extruder(764.48818)
  MoveL 1421 to (515.93, 549.41, 20) mm, rotated rx 180 ry 0 rz 160 deg; joints [11.939, 79.889, -19.402, -144.385, 65.289, 163.33]
  Set speed (17.5 mm/s)
  Call Extruder(768.04357)
  MoveL 1422 to (514.88, 549.73, 20) mm, rotated rx 180 ry 0 rz 160 deg; joints [12.003, 79.726, -19.032, -144.372, 65.476, 163.434]
  Set speed (17.5 mm/s)
  Call Extruder(771.49078)
  MoveL 1423 to (513.85, 550.03, 20) mm, rotated rx 180 ry 0 rz 160 deg; joints [12.065, 79.568, -18.673, -144.361, 65.657, 163.536]
  Set speed (17.5 mm/s)
  Call Extruder(774.36838)
  MoveL 1424 to (512.99, 550.26, 20) mm, rotated rx 180 ry 0 rz 160 deg; joints [12.113, 79.436, -18.37, -144.354, 65.808, 163.623]
  Set speed (17.5 mm/s)
  Call Extruder(778.29441)
  MoveL 1425 to (511.81, 550.55, 20) mm, rotated rx -180 ry 0 rz 160 deg; joints [12.178, 79.255, -17.958, -144.346, 66.015, 163.743]
  Set speed (17.5 mm/s)
  Call Extruder(785.18925)
  MoveL 1426 to (509.72, 550.99, 20) mm, rotated rx -180 ry 0 rz 160 deg; joints [12.285, 78.936, -17.228, -144.34, 66.379, 163.96]
  Set speed (17.5 mm/s)
  Call Extruder(792.11012)
  MoveL 1427 to (507.61, 551.35, 20) mm, rotated rx 180 ry 0 rz 160 deg; joints [12.383, 78.616, -16.491, -144.343, 66.744, 164.184]
  Set speed (17.5 mm/s)
  Call Extruder(798.87602)
  MoveL 1428 to (505.53, 551.62, 20) mm, rotated rx 180 ry 0 rz 160 deg; joints [12.469, 78.303, -15.769, -144.353, 67.1, 164.407]
  Set speed (17.5 mm/s)
  Call Extruder(805.77220)
  MoveL 1429 to (503.4, 551.8, 20) mm, rotated rx 180 ry 0 rz 160 deg; joints [12.548, 77.985, -15.032, -144.373, 67.462, 164.64]
  Set speed (17.5 mm/s)
  Call Extruder(812.67959)
  MoveL 1430 to (501.26, 551.9, 20) mm, rotated rx -180 ry 0 rz 160 deg; joints [12.618, 77.667, -14.292, -144.402, 67.823, 164.878]
  Set speed (17.5 mm/s)
  Call Extruder(819.43681)
  MoveL 1431 to (499.16, 551.9, 20) mm, rotated rx 180 ry 0 rz 160 deg; joints [12.676, 77.358, -13.57, -144.439, 68.174, 165.115]
  Set speed (10.0 mm/s)
  MoveL 1432 to (499.16, 551.9, 24) mm, rotated rx -180 ry 0 rz 160 deg; joints [12.676, 76.625, -13.023, -144.395, 68.023, 164.999]
  Set speed (120.0 mm/s)
  MoveL 1433 to (499.17, 552.87, 24) mm, rotated rx 180 ry 0 rz 160 deg; joints [12.793, 76.659, -13.102, -144.262, 68.017, 164.925]
  Set speed (17.5 mm/s)
  Call Extruder(826.56048)
  MoveL 1434 to (496.97, 552.79, 24) mm, rotated rx 180 ry 0 rz 160 deg; joints [12.845, 76.335, -12.344, -144.31, 68.382, 165.177]
  Call Extruder(833.57135)
  MoveL 1435 to (494.8, 552.62, 24) mm, rotated rx -180 ry 0 rz 160 deg; joints [12.885, 76.019, -11.602, -144.366, 68.738, 165.429]
  Set speed (17.5 mm/s)
  Call Extruder(840.47728)
  MoveL 1436 to (492.67, 552.37, 24) mm, rotated rx -180 ry 0 rz 160 deg; joints [12.913, 75.711, -10.876, -144.43, 69.086, 165.679]
  Set speed (17.5 mm/s)
  Call Extruder(847.34597)
  MoveL 1437 to (490.57, 552.03, 24) mm, rotated rx -180 ry 0 rz 160 deg; joints [12.931, 75.408, -10.158, -144.503, 69.428, 165.931]
  Set speed (17.5 mm/s)
  Call Extruder(854.52226)
  MoveL 1438 to (488.39, 551.59, 24) mm, rotated rx 180 ry 0 rz 160 deg; joints [12.938, 75.096, -9.414, -144.589, 69.781, 166.195]
  Set speed (17.5 mm/s)
  Call Extruder(857.92060)
  MoveL 1439 to (487.37, 551.35, 24) mm, rotated rx 180 ry 0 rz 160 deg; joints [12.937, 74.95, -9.065, -144.633, 69.946, 166.321]
  Set speed (17.5 mm/s)
  Call Extruder(861.29157)
  MoveL 1440 to (486.35, 551.09, 24) mm, rotated rx 180 ry 0 rz 160 deg; joints [12.934, 74.806, -8.72, -144.679, 70.109, 166.445]
  Set speed (17.5 mm/s)
  Call Extruder(863.41682)
  MoveL 1441 to (485.72, 550.91, 24) mm, rotated rx -180 ry 0 rz 160 deg; joints [12.931, 74.716, -8.504, -144.708, 70.211, 166.524]
  Set speed (17.5 mm/s)
  Call Extruder(868.53685)
  MoveL 1442 to (484.2, 550.47, 24) mm, rotated rx 180 ry 0 rz 160 deg; joints [12.918, 74.5, -7.986, -144.784, 70.455, 166.714]
  Set speed (17.5 mm/s)
  Call Extruder(875.33211)
  MoveL 1443 to (482.2, 549.8, 24) mm, rotated rx -180 ry 0 rz 160 deg; joints [12.891, 74.219, -7.306, -144.892, 70.775, 166.967]
  Set speed (17.5 mm/s)
  Call Extruder(882.17346)
  MoveL 1444 to (480.22, 549.04, 24) mm, rotated rx 180 ry 0 rz 160 deg; joints [12.853, 73.94, -6.63, -145.01, 71.092, 167.221]
  Set speed (17.5 mm/s)
  Call Extruder(885.86718)
  MoveL 1445 to (479.16, 548.6, 24) mm, rotated rx 180 ry 0 rz 160 deg; joints [12.827, 73.792, -6.27, -145.078, 71.261, 167.358]
  Set speed (17.5 mm/s)
  Call Extruder(889.19058)
  MoveL 1446 to (478.22, 548.19, 24) mm, rotated rx 180 ry 0 rz 160 deg; joints [12.802, 73.661, -5.948, -145.141, 71.411, 167.481]
  Set speed (17.5 mm/s)
  Call Extruder(892.96922)
  MoveL 1447 to (477.16, 547.69, 24) mm, rotated rx -180 ry 0 rz 160 deg; joints [12.77, 73.513, -5.585, -145.215, 71.58, 167.621]
  Set speed (17.5 mm/s)
  Call Extruder(898.02989)
  MoveL 1448 to (475.75, 547, 24) mm, rotated rx -180 ry 0 rz 160 deg; joints [12.722, 73.317, -5.106, -145.319, 71.803, 167.807]
  Call Extruder(903.78619)
  MoveL 1449 to (474.18, 546.15, 24) mm, rotated rx 180 ry 0 rz 160 deg; joints [12.658, 73.099, -4.569, -145.443, 72.053, 168.018]
  Set speed (17.5 mm/s)
  Call Extruder(906.67486)
  MoveL 1450 to (473.41, 545.71, 24) mm, rotated rx 180 ry 0 rz 160 deg; joints [12.624, 72.992, -4.302, -145.507, 72.177, 168.123]
  Set speed (17.5 mm/s)
  Call Extruder(910.22332)
  MoveL 1451 to (472.46, 545.14, 24) mm, rotated rx -180 ry 0 rz 160 deg; joints [12.578, 72.861, -3.978, -145.589, 72.327, 168.253]
  Set speed (17.5 mm/s)
  Call Extruder(913.65325)
  MoveL 1452 to (471.56, 544.58, 24) mm, rotated rx 180 ry 0 rz 160 deg; joints [12.531, 72.736, -3.668, -145.671, 72.47, 168.377]
  Set speed (17.5 mm/s)
  Call Extruder(917.25863)
  MoveL 1453 to (470.62, 543.97, 24) mm, rotated rx 180 ry 0 rz 160 deg; joints [12.479, 72.607, -3.346, -145.759, 72.619, 168.507]
  Set speed (17.5 mm/s)
  Call Extruder(920.60623)
  MoveL 1454 to (469.76, 543.38, 24) mm, rotated rx 180 ry 0 rz 160 deg; joints [12.427, 72.489, -3.051, -145.843, 72.755, 168.627]
  Set speed (17.5 mm/s)
  Call Extruder(924.13307)
  MoveL 1455 to (468.87, 542.75, 24) mm, rotated rx 180 ry 0 rz 160 deg; joints [12.37, 72.366, -2.744, -145.934, 72.896, 168.752]
  Set speed (17.5 mm/s)
  Call Extruder(927.75971)
  MoveL 1456 to (467.97, 542.08, 24) mm, rotated rx 180 ry 0 rz 160 deg; joints [12.308, 72.242, -2.432, -146.029, 73.04, 168.881]
  Set speed (17.5 mm/s)
  Call Extruder(931.15008)
  MoveL 1457 to (467.14, 541.43, 24) mm, rotated rx 180 ry 0 rz 160 deg; joints [12.247, 72.128, -2.145, -146.121, 73.172, 169]
  Set speed (17.5 mm/s)
  Call Extruder(934.63562)
  MoveL 1458 to (466.3, 540.75, 24) mm, rotated rx 180 ry 0 rz 160 deg; joints [12.181, 72.013, -1.855, -146.218, 73.305, 169.121]
  Set speed (17.5 mm/s)
  Call Extruder(938.21784)
  MoveL 1459 to (465.45, 540.04, 24) mm, rotated rx -180 ry 0 rz 160 deg; joints [12.111, 71.896, -1.559, -146.32, 73.44, 169.245]
  Set speed (17.5 mm/s)
  Call Extruder(941.57813)
  MoveL 1460 to (464.67, 539.35, 24) mm, rotated rx 180 ry 0 rz 160 deg; joints [12.042, 71.788, -1.287, -146.417, 73.565, 169.36]
  Set speed (17.5 mm/s)
  Call Extruder(945.08837)
  MoveL 1461 to (463.87, 538.61, 24) mm, rotated rx -180 ry 0 rz 160 deg; joints [11.967, 71.678, -1.007, -146.522, 73.692, 169.48]
  Set speed (17.5 mm/s)
  Call Extruder(948.56346)
  MoveL 1462 to (463.09, 537.87, 24) mm, rotated rx 180 ry 0 rz 160 deg; joints [11.89, 71.571, -0.735, -146.627, 73.816, 169.597]
  Call Extruder(952.05589)
  MoveL 1463 to (462.32, 537.1, 24) mm, rotated rx 180 ry 0 rz 160 deg; joints [11.81, 71.466, -0.465, -146.735, 73.939, 169.713]
  Set speed (17.5 mm/s)
  Call Extruder(955.52014)
  MoveL 1464 to (461.57, 536.33, 24) mm, rotated rx 180 ry 0 rz 160 deg; joints [11.727, 71.363, -0.203, -146.845, 74.058, 169.828]
  Call Extruder(959.04805)
  MoveL 1465 to (460.83, 535.53, 24) mm, rotated rx 180 ry 0 rz 160 deg; joints [11.64, 71.261, 0.059, -146.958, 74.177, 169.943]
  Set speed (17.5 mm/s)
  Call Extruder(962.48274)
  MoveL 1466 to (460.12, 534.73, 24) mm, rotated rx 180 ry 0 rz 160 deg; joints [11.553, 71.163, 0.31, -147.071, 74.29, 170.054]
  Set speed (17.5 mm/s)
  Call Extruder(966.03960)
  MoveL 1467 to (459.41, 533.89, 24) mm, rotated rx -180 ry 0 rz 160 deg; joints [11.46, 71.065, 0.565, -147.19, 74.405, 170.167]
  Call Extruder(969.50471)
  MoveL 1468 to (458.73, 533.06, 24) mm, rotated rx 180 ry 0 rz 160 deg; joints [11.366, 70.971, 0.807, -147.309, 74.514, 170.277]
  Set speed (17.5 mm/s)
  Call Extruder(975.04286)
  MoveL 1469 to (457.67, 531.71, 24) mm, rotated rx 180 ry 0 rz 160 deg; joints [11.211, 70.825, 1.185, -147.501, 74.684, 170.448]
  Set speed (17.5 mm/s)
  Call Extruder(979.97316)
  MoveL 1470 to (456.78, 530.47, 24) mm, rotated rx -180 ry 0 rz 160 deg; joints [11.067, 70.7, 1.509, -147.678, 74.828, 170.598]
  Set speed (17.5 mm/s)
  Call Extruder(983.49957)
  MoveL 1471 to (456.16, 529.57, 24) mm, rotated rx 180 ry 0 rz 160 deg; joints [10.961, 70.614, 1.734, -147.806, 74.928, 170.703]
  Set speed (17.5 mm/s)
  Call Extruder(986.97520)
  MoveL 1472 to (455.57, 528.67, 24) mm, rotated rx 180 ry 0 rz 160 deg; joints [10.854, 70.531, 1.951, -147.935, 75.024, 170.805]
  Call Extruder(990.43757)
  MoveL 1473 to (454.99, 527.76, 24) mm, rotated rx 180 ry 0 rz 160 deg; joints [10.745, 70.451, 2.161, -148.065, 75.117, 170.905]
  Set speed (17.5 mm/s)
  Call Extruder(993.94483)
  MoveL 1474 to (454.43, 526.83, 24) mm, rotated rx -180 ry 0 rz 160 deg; joints [10.632, 70.372, 2.369, -148.198, 75.208, 171.004]
  Set speed (17.5 mm/s)
  Call Extruder(999.57610)
  MoveL 1475 to (453.56, 525.31, 24) mm, rotated rx 180 ry 0 rz 160 deg; joints [10.445, 70.249, 2.692, -148.416, 75.35, 171.162]
  Set speed (17.5 mm/s)
  Call Extruder(1004.34335)
  MoveL 1476 to (452.88, 524, 24) mm, rotated rx 180 ry 0 rz 160 deg; joints [10.282, 70.151, 2.951, -148.605, 75.462, 171.29]
  Set speed (17.5 mm/s)
  Call Extruder(1007.81098)
  MoveL 1477 to (452.4, 523.03, 24) mm, rotated rx -180 ry 0 rz 160 deg; joints [10.161, 70.082, 3.133, -148.744, 75.541, 171.382]
  Set speed (17.5 mm/s)
  Call Extruder(1011.43849)
  MoveL 1478 to (451.93, 522.02, 24) mm, rotated rx -180 ry 0 rz 160 deg; joints [10.032, 70.013, 3.316, -148.891, 75.619, 171.476]
  Call Extruder(1015.01560)
  MoveL 1479 to (451.47, 521.01, 24) mm, rotated rx 180 ry 0 rz 160 deg; joints [9.903, 69.946, 3.492, -149.037, 75.694, 171.567]
  Set speed (17.5 mm/s)
  Call Extruder(1021.92576)
  MoveL 1480 to (450.66, 519.02, 24) mm, rotated rx -180 ry 0 rz 160 deg; joints [9.647, 69.826, 3.812, -149.324, 75.828, 171.737]
  Set speed (17.5 mm/s)
  Call Extruder(1028.73801)
  MoveL 1481 to (449.94, 517.04, 24) mm, rotated rx 180 ry 0 rz 160 deg; joints [9.387, 69.717, 4.104, -149.613, 75.948, 171.897]
  Set speed (17.5 mm/s)
  Call Extruder(1032.49116)
  MoveL 1482 to (449.58, 515.93, 24) mm, rotated rx -180 ry 0 rz 160 deg; joints [9.24, 69.661, 4.253, -149.774, 76.008, 171.982]
  Set speed (17.5 mm/s)
  Call Extruder(1035.74077)
  MoveL 1483 to (449.28, 514.97, 24) mm, rotated rx 180 ry 0 rz 160 deg; joints [9.112, 69.614, 4.378, -149.915, 76.058, 172.054]
  Set speed (17.5 mm/s)
  Call Extruder(1042.69747)
  MoveL 1484 to (448.72, 512.89, 24) mm, rotated rx -180 ry 0 rz 160 deg; joints [8.833, 69.522, 4.625, -150.219, 76.154, 172.202]
  Set speed (17.5 mm/s)
  Call Extruder(1045.73635)
  MoveL 1485 to (448.5, 511.97, 24) mm, rotated rx 180 ry 0 rz 160 deg; joints [8.709, 69.485, 4.724, -150.353, 76.192, 172.264]
  Set speed (17.5 mm/s)
  Call Extruder(1049.60496)
  MoveL 1486 to (448.24, 510.8, 24) mm, rotated rx -180 ry 0 rz 160 deg; joints [8.55, 69.44, 4.845, -150.525, 76.236, 172.341]
  Set speed (17.5 mm/s)
  Call Extruder(1056.82533)
  MoveL 1487 to (447.82, 508.6, 24) mm, rotated rx 180 ry 0 rz 160 deg; joints [8.248, 69.366, 5.047, -150.848, 76.307, 172.479]
  Set speed (17.5 mm/s)
  Call Extruder(1063.81841)
  MoveL 1488 to (447.52, 506.46, 24) mm, rotated rx 180 ry 0 rz 160 deg; joints [7.95, 69.303, 5.215, -151.164, 76.362, 172.603]
  Set speed (17.5 mm/s)
  Call Extruder(1070.79812)
  MoveL 1489 to (447.3, 504.3, 24) mm, rotated rx 180 ry 0 rz 160 deg; joints [7.649, 69.251, 5.357, -151.482, 76.401, 172.72]
  Set speed (17.5 mm/s)
  Call Extruder(1077.59235)
  MoveL 1490 to (447.16, 502.2, 24) mm, rotated rx -180 ry 0 rz 160 deg; joints [7.353, 69.21, 5.468, -151.792, 76.426, 172.825]
  Set speed (17.5 mm/s)
  Call Extruder(1084.65688)
  MoveL 1491 to (447.12, 500.01, 24) mm, rotated rx 180 ry 0 rz 160 deg; joints [7.042, 69.177, 5.556, -152.115, 76.437, 172.926]
  Set speed (17.5 mm/s)
  Call Extruder(1091.01512)
  MoveL 1492 to (447.15, 498.04, 24) mm, rotated rx 180 ry 0 rz 160 deg; joints [6.761, 69.157, 5.612, -152.406, 76.433, 173.01]
  Call Extruder(1097.14303)
  MoveL 1493 to (447.26, 496.14, 24) mm, rotated rx -180 ry 0 rz 160 deg; joints [6.489, 69.145, 5.643, -152.687, 76.418, 173.085]
  Set speed (17.5 mm/s)
  Call Extruder(1103.49292)
  MoveL 1494 to (447.44, 494.19, 24) mm, rotated rx 180 ry 0 rz 160 deg; joints [6.206, 69.142, 5.654, -152.976, 76.39, 173.156]
  Set speed (17.5 mm/s)
  Call Extruder(1109.77189)
  MoveL 1495 to (447.69, 492.25, 24) mm, rotated rx -180 ry 0 rz 160 deg; joints [5.927, 69.146, 5.641, -153.261, 76.35, 173.22]
  Set speed (17.5 mm/s)
  Call Extruder(1115.88410)
  MoveL 1496 to (448, 490.38, 24) mm, rotated rx 180 ry 0 rz 160 deg; joints [5.655, 69.158, 5.608, -153.536, 76.299, 173.276]
  Set speed (17.5 mm/s)
  Call Extruder(1122.26414)
  MoveL 1497 to (448.4, 488.44, 24) mm, rotated rx -180 ry 0 rz 160 deg; joints [5.373, 69.179, 5.551, -153.821, 76.234, 173.328]
  Set speed (17.5 mm/s)
  Call Extruder(1128.63884)
  MoveL 1498 to (448.87, 486.52, 24) mm, rotated rx 180 ry 0 rz 160 deg; joints [5.092, 69.209, 5.47, -154.102, 76.156, 173.373]
  Set speed (17.5 mm/s)
  Call Extruder(1134.87677)
  MoveL 1499 to (449.39, 484.66, 24) mm, rotated rx -180 ry 0 rz 160 deg; joints [4.82, 69.246, 5.37, -154.374, 76.067, 173.412]
  Call Extruder(1141.09003)
  MoveL 1500 to (449.99, 482.83, 24) mm, rotated rx 180 ry 0 rz 160 deg; joints [4.551, 69.291, 5.248, -154.641, 75.967, 173.444]
  Set speed (17.5 mm/s)
  Call Extruder(1147.50044)
  MoveL 1501 to (450.67, 480.96, 24) mm, rotated rx -180 ry 0 rz 160 deg; joints [4.278, 69.346, 5.1, -154.911, 75.851, 173.471]
  Set speed (17.5 mm/s)
  Call Extruder(1153.79361)
  MoveL 1502 to (451.4, 479.15, 24) mm, rotated rx 180 ry 0 rz 160 deg; joints [4.013, 69.408, 4.932, -155.171, 75.726, 173.492]
  Set speed (17.5 mm/s)
  Call Extruder(1160.07652)
  MoveL 1503 to (452.2, 477.37, 24) mm, rotated rx -180 ry 0 rz 160 deg; joints [3.752, 69.478, 4.744, -155.426, 75.589, 173.507]
  Set speed (17.5 mm/s)
  Call Extruder(1166.21648)
  MoveL 1504 to (453.05, 475.67, 24) mm, rotated rx 180 ry 0 rz 160 deg; joints [3.503, 69.554, 4.539, -155.668, 75.443, 173.516]
  Call Extruder(1172.53589)
  MoveL 1505 to (453.98, 473.95, 24) mm, rotated rx 180 ry 0 rz 160 deg; joints [3.251, 69.641, 4.307, -155.911, 75.282, 173.52]
  Set speed (17.5 mm/s)
  Call Extruder(1178.74825)
  MoveL 1506 to (454.96, 472.29, 24) mm, rotated rx -180 ry 0 rz 160 deg; joints [3.009, 69.734, 4.058, -156.143, 75.112, 173.518]
  Call Extruder(1185.10089)
  MoveL 1507 to (456.02, 470.63, 24) mm, rotated rx -180 ry 0 rz 160 deg; joints [2.767, 69.837, 3.783, -156.374, 74.928, 173.51]
  Set speed (17.5 mm/s)
  Call Extruder(1191.36872)
  MoveL 1508 to (457.13, 469.04, 24) mm, rotated rx 180 ry 0 rz 160 deg; joints [2.535, 69.946, 3.492, -156.593, 74.735, 173.498]
  Set speed (17.5 mm/s)
  Call Extruder(1197.74520)
  MoveL 1509 to (458.32, 467.46, 24) mm, rotated rx 180 ry 0 rz 160 deg; joints [2.306, 70.066, 3.175, -156.807, 74.528, 173.48]
  Set speed (17.5 mm/s)
  Call Extruder(1203.93777)
  MoveL 1510 to (459.53, 465.96, 24) mm, rotated rx 180 ry 0 rz 160 deg; joints [2.09, 70.189, 2.848, -157.008, 74.316, 173.456]
  Call Extruder(1210.22310)
  MoveL 1511 to (460.81, 464.5, 24) mm, rotated rx -180 ry 0 rz 160 deg; joints [1.879, 70.322, 2.498, -157.202, 74.092, 173.428]
  Set speed (17.5 mm/s)
  Call Extruder(1216.58013)
  MoveL 1512 to (462.16, 463.06, 24) mm, rotated rx -180 ry 0 rz 160 deg; joints [1.673, 70.465, 2.124, -157.389, 73.855, 173.394]
  Call Extruder(1222.77462)
  MoveL 1513 to (463.53, 461.71, 24) mm, rotated rx -180 ry 0 rz 160 deg; joints [1.48, 70.611, 1.742, -157.562, 73.615, 173.355]
  Call Extruder(1228.89002)
  MoveL 1514 to (464.92, 460.43, 24) mm, rotated rx -180 ry 0 rz 160 deg; joints [1.298, 70.762, 1.348, -157.724, 73.369, 173.313]
  Set speed (17.5 mm/s)
  Call Extruder(1235.41486)
  MoveL 1515 to (466.46, 459.12, 24) mm, rotated rx 180 ry 0 rz 160 deg; joints [1.112, 70.932, 0.909, -157.885, 73.097, 173.262]
  Set speed (17.5 mm/s)
  Call Extruder(1241.54573)
  MoveL 1516 to (467.95, 457.94, 24) mm, rotated rx -180 ry 0 rz 160 deg; joints [0.946, 71.098, 0.48, -158.027, 72.834, 173.209]
  Set speed (17.5 mm/s)
  Call Extruder(1247.96911)
  MoveL 1517 to (469.56, 456.76, 24) mm, rotated rx -180 ry 0 rz 160 deg; joints [0.782, 71.279, 0.013, -158.165, 72.55, 173.149]
  Set speed (17.5 mm/s)
  Call Extruder(1254.16408)
  MoveL 1518 to (471.15, 455.68, 24) mm, rotated rx -180 ry 0 rz 160 deg; joints [0.632, 71.461, -0.452, -158.288, 72.269, 173.085]
  Set speed (17.5 mm/s)
  Call Extruder(1260.53917)
  MoveL 1519 to (472.83, 454.64, 24) mm, rotated rx -180 ry 0 rz 160 deg; joints [0.488, 71.655, -0.947, -158.403, 71.972, 173.015]
  Set speed (17.5 mm/s)
  Call Extruder(1266.80252)
  MoveL 1520 to (474.51, 453.67, 24) mm, rotated rx 180 ry 0 rz 160 deg; joints [0.355, 71.852, -1.448, -158.505, 71.673, 172.941]
  Set speed (17.5 mm/s)
  Call Extruder(1273.05426)
  MoveL 1521 to (476.23, 452.76, 24) mm, rotated rx -180 ry 0 rz 160 deg; joints [0.232, 72.055, -1.962, -158.596, 71.368, 172.862]
  Set speed (17.5 mm/s)
  Call Extruder(1279.17069)
  MoveL 1522 to (477.93, 451.94, 24) mm, rotated rx -180 ry 0 rz 160 deg; joints [0.121, 72.26, -2.478, -158.674, 71.065, 172.78]
  Set speed (17.5 mm/s)
  Call Extruder(1285.65147)
  MoveL 1523 to (479.78, 451.14, 24) mm, rotated rx 180 ry 0 rz 160 deg; joints [0.013, 72.484, -3.038, -158.745, 70.737, 172.687]
  Set speed (17.5 mm/s)
  Call Extruder(1291.83143)
  MoveL 1524 to (481.56, 450.44, 24) mm, rotated rx -180 ry 0 rz 160 deg; joints [-0.08, 72.703, -3.586, -158.801, 70.42, 172.594]
  Set speed (17.5 mm/s)
  Call Extruder(1298.18731)
  MoveL 1525 to (483.42, 449.79, 24) mm, rotated rx -180 ry 0 rz 160 deg; joints [-0.166, 72.935, -4.161, -158.847, 70.088, 172.493]
  Set speed (17.5 mm/s)
  Call Extruder(1304.33103)
  MoveL 1526 to (485.24, 449.22, 24) mm, rotated rx -180 ry 0 rz 160 deg; joints [-0.24, 73.164, -4.728, -158.88, 69.764, 172.39]
  Set speed (17.5 mm/s)
  Call Extruder(1310.67182)
  MoveL 1527 to (487.14, 448.71, 24) mm, rotated rx 180 ry 0 rz 160 deg; joints [-0.306, 73.406, -5.323, -158.903, 69.425, 172.278]
  Set speed (17.5 mm/s)
  Call Extruder(1317.03938)
  MoveL 1528 to (489.06, 448.26, 24) mm, rotated rx 180 ry 0 rz 160 deg; joints [-0.363, 73.654, -5.932, -158.914, 69.081, 172.161]
  Set speed (17.5 mm/s)
  Call Extruder(1323.24496)
  MoveL 1529 to (490.95, 447.9, 24) mm, rotated rx 180 ry 0 rz 160 deg; joints [-0.409, 73.901, -6.535, -158.913, 68.743, 172.041]
  Set speed (17.5 mm/s)
  Call Extruder(1329.17280)
  MoveL 1530 to (492.77, 447.62, 24) mm, rotated rx 180 ry 0 rz 160 deg; joints [-0.444, 74.141, -7.118, -158.902, 68.417, 171.922]
  Set speed (17.5 mm/s)
  Call Extruder(1335.67204)
  MoveL 1531 to (494.77, 447.38, 24) mm, rotated rx -180 ry 0 rz 160 deg; joints [-0.472, 74.409, -7.767, -158.878, 68.058, 171.786]
  Call Extruder(1342.01231)
  MoveL 1532 to (496.73, 447.22, 24) mm, rotated rx 180 ry 0 rz 160 deg; joints [-0.491, 74.675, -8.407, -158.842, 67.707, 171.648]
  Call Extruder(1348.43821)
  MoveL 1533 to (498.71, 447.14, 24) mm, rotated rx 180 ry 0 rz 160 deg; joints [-0.5, 74.949, -9.063, -158.795, 67.349, 171.502]
  Set speed (17.5 mm/s)
  Call Extruder(1354.64598)
  MoveL 1534 to (500.64, 447.12, 24) mm, rotated rx -180 ry 0 rz 160 deg; joints [-0.499, 75.217, -9.703, -158.737, 67.002, 171.355]
  Set speed (17.5 mm/s)
  Call Extruder(1360.99601)
  MoveL 1535 to (502.61, 447.18, 24) mm, rotated rx 180 ry 0 rz 160 deg; joints [-0.489, 75.495, -10.364, -158.667, 66.647, 171.2]
  Set speed (17.5 mm/s)
  Call Extruder(1367.19166)
  MoveL 1536 to (504.53, 447.31, 24) mm, rotated rx 180 ry 0 rz 160 deg; joints [-0.471, 75.769, -11.013, -158.588, 66.301, 171.043]
  Set speed (17.5 mm/s)
  Call Extruder(1373.34173)
  MoveL 1537 to (506.42, 447.51, 24) mm, rotated rx -180 ry 0 rz 160 deg; joints [-0.444, 76.044, -11.661, -158.498, 65.958, 170.882]
  Set speed (17.5 mm/s)
  Call Extruder(1379.66215)
  MoveL 1538 to (508.37, 447.79, 24) mm, rotated rx 180 ry 0 rz 160 deg; joints [-0.408, 76.329, -12.33, -158.396, 65.606, 170.711]
  Call Extruder(1386.10023)
  MoveL 1539 to (510.33, 448.14, 24) mm, rotated rx -180 ry 0 rz 160 deg; joints [-0.362, 76.621, -13.014, -158.28, 65.25, 170.532]
  Call Extruder(1392.31856)
  MoveL 1540 to (512.21, 448.55, 24) mm, rotated rx -180 ry 0 rz 160 deg; joints [-0.309, 76.906, -13.676, -158.158, 64.908, 170.353]
  Set speed (17.5 mm/s)
  Call Extruder(1398.49540)
  MoveL 1541 to (514.07, 449.02, 24) mm, rotated rx -180 ry 0 rz 160 deg; joints [-0.25, 77.19, -14.335, -158.026, 64.57, 170.171]
  Call Extruder(1404.85613)
  MoveL 1542 to (515.96, 449.58, 24) mm, rotated rx 180 ry 0 rz 160 deg; joints [-0.18, 77.483, -15.013, -157.881, 64.225, 169.977]
  Set speed (17.5 mm/s)
  Call Extruder(1411.20579)
  MoveL 1543 to (517.83, 450.22, 24) mm, rotated rx -180 ry 0 rz 160 deg; joints [-0.102, 77.777, -15.69, -157.725, 63.885, 169.779]
  Call Extruder(1417.38837)
  MoveL 1544 to (519.62, 450.9, 24) mm, rotated rx -180 ry 0 rz 160 deg; joints [-0.018, 78.063, -16.347, -157.564, 63.557, 169.581]
  Call Extruder(1423.75656)
  MoveL 1545 to (521.44, 451.66, 24) mm, rotated rx 180 ry 0 rz 160 deg; joints [0.075, 78.358, -17.021, -157.388, 63.224, 169.373]
  Set speed (17.5 mm/s)
  Call Extruder(1429.80553)
  MoveL 1546 to (523.14, 452.45, 24) mm, rotated rx 180 ry 0 rz 160 deg; joints [0.171, 78.638, -17.659, -157.213, 62.911, 169.17]
  Set speed (17.5 mm/s)
  Call Extruder(1436.32466)
  MoveL 1547 to (524.95, 453.37, 24) mm, rotated rx 180 ry 0 rz 160 deg; joints [0.282, 78.939, -18.341, -157.014, 62.581, 168.947]
  Set speed (17.5 mm/s)
  Call Extruder(1442.58115)
  MoveL 1548 to (526.64, 454.32, 24) mm, rotated rx -180 ry 0 rz 160 deg; joints [0.394, 79.226, -18.991, -156.815, 62.269, 168.729]
  Set speed (17.5 mm/s)
  Call Extruder(1448.76518)
  MoveL 1549 to (528.28, 455.32, 24) mm, rotated rx -180 ry 0 rz 160 deg; joints [0.513, 79.508, -19.628, -156.61, 61.967, 168.509]
  Call Extruder(1455.13973)
  MoveL 1550 to (529.93, 456.41, 24) mm, rotated rx -180 ry 0 rz 160 deg; joints [0.641, 79.797, -20.276, -156.39, 61.662, 168.279]
  Set speed (17.5 mm/s)
  Call Extruder(1461.25881)
  MoveL 1551 to (531.47, 457.51, 24) mm, rotated rx -180 ry 0 rz 160 deg; joints [0.77, 80.071, -20.891, -156.172, 61.377, 168.054]
  Call Extruder(1467.60369)
  MoveL 1552 to (533.03, 458.71, 24) mm, rotated rx 180 ry 0 rz 160 deg; joints [0.91, 80.352, -21.519, -155.938, 61.089, 167.818]
  Set speed (17.5 mm/s)
  Call Extruder(1473.88046)
  MoveL 1553 to (534.53, 459.95, 24) mm, rotated rx -180 ry 0 rz 160 deg; joints [1.055, 80.627, -22.132, -155.7, 60.812, 167.582]
  Call Extruder(1480.24955)
  MoveL 1554 to (536, 461.27, 24) mm, rotated rx -180 ry 0 rz 160 deg; joints [1.207, 80.902, -22.742, -155.451, 60.539, 167.339]
  Set speed (17.5 mm/s)
  Call Extruder(1486.29211)
  MoveL 1555 to (537.35, 462.57, 24) mm, rotated rx 180 ry 0 rz 160 deg; joints [1.357, 81.158, -23.31, -155.21, 60.289, 167.107]
  Set speed (17.5 mm/s)
  Call Extruder(1489.90736)
  MoveL 1556 to (538.14, 463.37, 24) mm, rotated rx -180 ry 0 rz 160 deg; joints [1.449, 81.309, -23.643, -155.063, 60.144, 166.967]
  Set speed (17.5 mm/s)
  Call Extruder(1493.54531)
  MoveL 1557 to (538.91, 464.19, 24) mm, rotated rx -180 ry 0 rz 160 deg; joints [1.543, 81.46, -23.976, -154.913, 60.001, 166.826]
  Set speed (17.5 mm/s)
  Call Extruder(1496.89374)
  MoveL 1558 to (539.61, 464.96, 24) mm, rotated rx 180 ry 0 rz 160 deg; joints [1.631, 81.596, -24.277, -154.773, 59.872, 166.695]
  Set speed (17.5 mm/s)
  Call Extruder(1500.31697)
  MoveL 1559 to (540.3, 465.77, 24) mm, rotated rx -180 ry 0 rz 160 deg; joints [1.723, 81.733, -24.579, -154.629, 59.744, 166.562]
  Set speed (17.5 mm/s)
  Call Extruder(1503.82170)
  MoveL 1560 to (541, 466.6, 24) mm, rotated rx 180 ry 0 rz 160 deg; joints [1.818, 81.873, -24.886, -154.48, 59.615, 166.425]
  Set speed (17.5 mm/s)
  Call Extruder(1507.27035)
  MoveL 1561 to (541.66, 467.44, 24) mm, rotated rx -180 ry 0 rz 160 deg; joints [1.913, 82.008, -25.182, -154.332, 59.492, 166.289]
  Set speed (17.5 mm/s)
  Call Extruder(1510.78087)
  MoveL 1562 to (542.33, 468.3, 24) mm, rotated rx 180 ry 0 rz 160 deg; joints [2.011, 82.143, -25.479, -154.18, 59.37, 166.152]
  Set speed (17.5 mm/s)
  Call Extruder(1513.68308)
  MoveL 1563 to (542.86, 469.03, 24) mm, rotated rx -180 ry 0 rz 160 deg; joints [2.093, 82.253, -25.72, -154.053, 59.272, 166.038]
  Set speed (17.5 mm/s)
  Call Extruder(1517.70818)
  MoveL 1564 to (543.58, 470.05, 24) mm, rotated rx -180 ry 0 rz 160 deg; joints [2.208, 82.403, -26.048, -153.876, 59.14, 165.88]
  Set speed (17.5 mm/s)
  Call Extruder(1521.24996)
  MoveL 1565 to (544.19, 470.96, 24) mm, rotated rx 180 ry 0 rz 160 deg; joints [2.311, 82.532, -26.331, -153.719, 59.028, 165.741]
  Set speed (17.5 mm/s)
  Call Extruder(1524.70774)
  MoveL 1566 to (544.77, 471.86, 24) mm, rotated rx -180 ry 0 rz 160 deg; joints [2.413, 82.656, -26.601, -153.565, 58.922, 165.606]
  Set speed (17.5 mm/s)
  Call Extruder(1528.25592)
  MoveL 1567 to (545.35, 472.8, 24) mm, rotated rx -180 ry 0 rz 160 deg; joints [2.518, 82.781, -26.873, -153.406, 58.816, 165.468]
  Set speed (17.5 mm/s)
  Call Extruder(1531.68276)
  MoveL 1568 to (545.89, 473.71, 24) mm, rotated rx -180 ry 0 rz 160 deg; joints [2.621, 82.899, -27.129, -153.252, 58.719, 165.335]
  Set speed (17.5 mm/s)
  Call Extruder(1537.32475)
  MoveL 1569 to (546.73, 475.25, 24) mm, rotated rx 180 ry 0 rz 160 deg; joints [2.793, 83.086, -27.537, -152.996, 58.566, 165.117]
  Set speed (17.5 mm/s)
  Call Extruder(1542.25719)
  MoveL 1570 to (547.43, 476.61, 24) mm, rotated rx 180 ry 0 rz 160 deg; joints [2.946, 83.244, -27.881, -152.772, 58.44, 164.927]
  Set speed (17.5 mm/s)
  Call Extruder(1545.66499)
  MoveL 1571 to (547.88, 477.56, 24) mm, rotated rx -180 ry 0 rz 160 deg; joints [3.053, 83.35, -28.109, -152.616, 58.359, 164.797]
  Set speed (17.5 mm/s)
  Call Extruder(1549.23892)
  MoveL 1572 to (548.34, 478.57, 24) mm, rotated rx -180 ry 0 rz 160 deg; joints [3.166, 83.457, -28.342, -152.452, 58.277, 164.662]
  Set speed (17.5 mm/s)
  Call Extruder(1556.05681)
  MoveL 1573 to (549.16, 480.52, 24) mm, rotated rx 180 ry 0 rz 160 deg; joints [3.384, 83.653, -28.765, -152.139, 58.134, 164.407]
  Set speed (17.5 mm/s)
  Call Extruder(1559.69115)
  MoveL 1574 to (549.56, 481.57, 24) mm, rotated rx -180 ry 0 rz 160 deg; joints [3.502, 83.751, -28.977, -151.972, 58.065, 164.274]
  Call Extruder(1563.14909)
  MoveL 1575 to (549.93, 482.58, 24) mm, rotated rx -180 ry 0 rz 160 deg; joints [3.614, 83.843, -29.175, -151.813, 58.002, 164.147]
  Set speed (17.5 mm/s)
  Call Extruder(1570.32997)
  MoveL 1576 to (550.62, 484.69, 24) mm, rotated rx -180 ry 0 rz 160 deg; joints [3.851, 84.021, -29.56, -151.484, 57.885, 163.889]
  Call Extruder(0.00000)
  Call Extruder(6.60014)
  MoveL 1577 to (551.17, 486.66, 24) mm, rotated rx 180 ry 0 rz 160 deg; joints [4.071, 84.17, -29.881, -151.182, 57.796, 163.659]
  Set speed (17.5 mm/s)
  Call Extruder(10.29686)
  MoveL 1578 to (551.44, 487.78, 24) mm, rotated rx -180 ry 0 rz 160 deg; joints [4.196, 84.247, -30.047, -151.014, 57.753, 163.533]
  Call Extruder(13.72704)
  MoveL 1579 to (551.68, 488.81, 24) mm, rotated rx 180 ry 0 rz 160 deg; joints [4.311, 84.317, -30.196, -150.858, 57.717, 163.417]
  Set speed (17.5 mm/s)
  Call Extruder(20.73231)
  MoveL 1580 to (552.1, 490.94, 24) mm, rotated rx -180 ry 0 rz 160 deg; joints [4.55, 84.444, -30.47, -150.542, 57.657, 163.187]
  Set speed (17.5 mm/s)
  Call Extruder(27.64635)
  MoveL 1581 to (552.42, 493.06, 24) mm, rotated rx -180 ry 0 rz 160 deg; joints [4.788, 84.554, -30.706, -150.234, 57.617, 162.97]
  Set speed (17.5 mm/s)
  Call Extruder(34.78111)
  MoveL 1582 to (552.67, 495.26, 24) mm, rotated rx -180 ry 0 rz 160 deg; joints [5.035, 84.65, -30.912, -149.92, 57.595, 162.755]
  Set speed (17.5 mm/s)
  Call Extruder(41.66207)
  MoveL 1583 to (552.82, 497.39, 24) mm, rotated rx 180 ry 0 rz 160 deg; joints [5.274, 84.726, -31.075, -149.621, 57.591, 162.558]
  Call Extruder(48.63891)
  MoveL 1584 to (552.88, 499.56, 24) mm, rotated rx 180 ry 0 rz 160 deg; joints [5.518, 84.786, -31.204, -149.323, 57.605, 162.369]
  Set speed (17.5 mm/s)
  Call Extruder(55.69243)
  MoveL 1585 to (552.85, 501.74, 24) mm, rotated rx 180 ry 0 rz 160 deg; joints [5.766, 84.829, -31.295, -149.028, 57.639, 162.19]
  Set speed (17.5 mm/s)
  Call Extruder(62.57000)
  MoveL 1586 to (552.74, 503.87, 24) mm, rotated rx 180 ry 0 rz 160 deg; joints [6.007, 84.852, -31.345, -148.747, 57.69, 162.028]
  Set speed (17.5 mm/s)
  Call Extruder(69.55061)
  MoveL 1587 to (552.53, 506.03, 24) mm, rotated rx -180 ry 0 rz 160 deg; joints [6.253, 84.859, -31.358, -148.468, 57.76, 161.876]
  Set speed (17.5 mm/s)
  Call Extruder(76.61860)
  MoveL 1588 to (552.24, 508.2, 24) mm, rotated rx 180 ry 0 rz 160 deg; joints [6.502, 84.847, -31.333, -148.194, 57.85, 161.736]
  Set speed (17.5 mm/s)
  Call Extruder(83.56790)
  MoveL 1589 to (551.86, 510.32, 24) mm, rotated rx 180 ry 0 rz 160 deg; joints [6.746, 84.817, -31.27, -147.931, 57.955, 161.611]
  Set speed (17.5 mm/s)
  Call Extruder(90.83800)
  MoveL 1590 to (551.38, 512.52, 24) mm, rotated rx 180 ry 0 rz 160 deg; joints [7.001, 84.768, -31.165, -147.665, 58.083, 161.496]
  Call Extruder(97.42503)
  MoveL 1591 to (550.85, 514.5, 24) mm, rotated rx -180 ry 0 rz 160 deg; joints [7.231, 84.707, -31.034, -147.432, 58.215, 161.404]
  Set speed (17.5 mm/s)
  Call Extruder(104.34052)
  MoveL 1592 to (550.22, 516.55, 24) mm, rotated rx 180 ry 0 rz 160 deg; joints [7.471, 84.626, -30.859, -147.195, 58.37, 161.323]
  Call Extruder(111.27246)
  MoveL 1593 to (549.51, 518.58, 24) mm, rotated rx -180 ry 0 rz 160 deg; joints [7.711, 84.528, -30.649, -146.966, 58.541, 161.255]
  Set speed (17.5 mm/s)
  Call Extruder(114.89964)
  MoveL 1594 to (549.1, 519.62, 24) mm, rotated rx -180 ry 0 rz 160 deg; joints [7.835, 84.469, -30.523, -146.851, 58.637, 161.226]
  Set speed (17.5 mm/s)
  Call Extruder(118.26652)
  MoveL 1595 to (548.71, 520.59, 24) mm, rotated rx -180 ry 0 rz 160 deg; joints [7.95, 84.412, -30.401, -146.745, 58.729, 161.202]
  Set speed (17.5 mm/s)
  Call Extruder(120.57600)
  MoveL 1596 to (548.42, 521.25, 24) mm, rotated rx -180 ry 0 rz 160 deg; joints [8.029, 84.37, -30.311, -146.674, 58.795, 161.187]
  Set speed (17.5 mm/s)
  Call Extruder(127.02363)
  MoveL 1597 to (547.59, 523.06, 24) mm, rotated rx 180 ry 0 rz 160 deg; joints [8.247, 84.246, -30.044, -146.48, 58.984, 161.155]
  Set speed (17.5 mm/s)
  Call Extruder(132.37678)
  MoveL 1598 to (546.84, 524.54, 24) mm, rotated rx 180 ry 0 rz 160 deg; joints [8.427, 84.132, -29.798, -146.326, 59.152, 161.138]
  Set speed (17.5 mm/s)
  Call Extruder(135.86927)
  MoveL 1599 to (546.33, 525.49, 24) mm, rotated rx 180 ry 0 rz 160 deg; joints [8.543, 84.052, -29.626, -146.228, 59.266, 161.132]
  Set speed (17.5 mm/s)
  Call Extruder(139.34038)
  MoveL 1600 to (545.8, 526.43, 24) mm, rotated rx 180 ry 0 rz 160 deg; joints [8.658, 83.969, -29.448, -146.133, 59.383, 161.129]
  Set speed (17.5 mm/s)
  Call Extruder(142.86249)
  MoveL 1601 to (545.25, 527.37, 24) mm, rotated rx 180 ry 0 rz 160 deg; joints [8.774, 83.881, -29.259, -146.039, 59.505, 161.13]
  Set speed (17.5 mm/s)
  Call Extruder(145.57086)
  MoveL 1602 to (544.81, 528.09, 24) mm, rotated rx 180 ry 0 rz 160 deg; joints [8.863, 83.812, -29.109, -145.968, 59.6, 161.133]
  Set speed (17.5 mm/s)
  Call Extruder(150.34994)
  MoveL 1603 to (544, 529.33, 24) mm, rotated rx 180 ry 0 rz 160 deg; joints [9.018, 83.683, -28.831, -145.846, 59.774, 161.144]
  Call Extruder(153.29377)
  MoveL 1604 to (543.49, 530.09, 24) mm, rotated rx -180 ry 0 rz 160 deg; joints [9.113, 83.602, -28.654, -145.773, 59.883, 161.153]
  Set speed (17.5 mm/s)
  Call Extruder(156.71973)
  MoveL 1605 to (542.87, 530.96, 24) mm, rotated rx 180 ry 0 rz 160 deg; joints [9.223, 83.503, -28.44, -145.691, 60.014, 161.168]
  Set speed (17.5 mm/s)
  Call Extruder(160.18446)
  MoveL 1606 to (542.24, 531.82, 24) mm, rotated rx -180 ry 0 rz 160 deg; joints [9.333, 83.4, -28.217, -145.61, 60.148, 161.186]
  Set speed (17.5 mm/s)
  Call Extruder(163.75198)
  MoveL 1607 to (541.56, 532.7, 24) mm, rotated rx -180 ry 0 rz 160 deg; joints [9.445, 83.29, -27.98, -145.529, 60.29, 161.209]
  Set speed (17.5 mm/s)
  Call Extruder(167.16606)
  MoveL 1608 to (540.9, 533.52, 24) mm, rotated rx -180 ry 0 rz 160 deg; joints [9.551, 83.183, -27.748, -145.453, 60.427, 161.233]
  Set speed (17.5 mm/s)
  Call Extruder(170.70672)
  MoveL 1609 to (540.19, 534.37, 24) mm, rotated rx -180 ry 0 rz 160 deg; joints [9.661, 83.069, -27.498, -145.377, 60.573, 161.262]
  Set speed (17.5 mm/s)
  Call Extruder(174.14373)
  MoveL 1610 to (539.49, 535.17, 24) mm, rotated rx 180 ry 0 rz 160 deg; joints [9.766, 82.955, -27.251, -145.306, 60.717, 161.293]
  Set speed (17.5 mm/s)
  Call Extruder(177.62555)
  MoveL 1611 to (538.76, 535.97, 24) mm, rotated rx 180 ry 0 rz 160 deg; joints [9.871, 82.836, -26.993, -145.236, 60.865, 161.328]
  Set speed (17.5 mm/s)
  Call Extruder(180.41332)
  MoveL 1612 to (538.17, 536.6, 24) mm, rotated rx 180 ry 0 rz 160 deg; joints [9.955, 82.74, -26.784, -145.181, 60.985, 161.358]
  Call Extruder(184.65117)
  MoveL 1613 to (537.25, 537.53, 24) mm, rotated rx -180 ry 0 rz 160 deg; joints [10.08, 82.59, -26.457, -145.102, 61.17, 161.408]
  Set speed (17.5 mm/s)
  Call Extruder(188.08850)
  MoveL 1614 to (536.49, 538.28, 24) mm, rotated rx 180 ry 0 rz 160 deg; joints [10.18, 82.466, -26.185, -145.039, 61.323, 161.452]
  Call Extruder(191.58233)
  MoveL 1615 to (535.7, 539.02, 24) mm, rotated rx 180 ry 0 rz 160 deg; joints [10.281, 82.337, -25.903, -144.978, 61.48, 161.5]
  Set speed (17.5 mm/s)
  Call Extruder(194.35146)
  MoveL 1616 to (535.06, 539.59, 24) mm, rotated rx 180 ry 0 rz 160 deg; joints [10.36, 82.233, -25.676, -144.932, 61.606, 161.54]
  Call Extruder(198.55824)
  MoveL 1617 to (534.07, 540.44, 24) mm, rotated rx 180 ry 0 rz 160 deg; joints [10.479, 82.073, -25.325, -144.863, 61.8, 161.604]
  Set speed (17.5 mm/s)
  Call Extruder(202.07873)
  MoveL 1618 to (533.23, 541.14, 24) mm, rotated rx 180 ry 0 rz 160 deg; joints [10.576, 81.936, -25.024, -144.808, 61.964, 161.662]
  Call Extruder(205.50672)
  MoveL 1619 to (532.4, 541.8, 24) mm, rotated rx -180 ry 0 rz 160 deg; joints [10.67, 81.801, -24.728, -144.757, 62.126, 161.72]
  Set speed (17.5 mm/s)
  Call Extruder(209.02952)
  MoveL 1620 to (531.53, 542.46, 24) mm, rotated rx 180 ry 0 rz 160 deg; joints [10.765, 81.66, -24.418, -144.707, 62.294, 161.783]
  Call Extruder(212.57137)
  MoveL 1621 to (530.64, 543.1, 24) mm, rotated rx 180 ry 0 rz 160 deg; joints [10.859, 81.516, -24.101, -144.659, 62.464, 161.849]
  Set speed (17.5 mm/s)
  Call Extruder(216.05052)
  MoveL 1622 to (529.75, 543.72, 24) mm, rotated rx -180 ry 0 rz 160 deg; joints [10.949, 81.374, -23.786, -144.613, 62.633, 161.917]
  Set speed (17.5 mm/s)
  Call Extruder(220.19466)
  MoveL 1623 to (528.68, 544.43, 24) mm, rotated rx -180 ry 0 rz 160 deg; joints [11.055, 81.201, -23.405, -144.562, 62.835, 162.001]
  Set speed (17.5 mm/s)
  Call Extruder(226.41315)
  MoveL 1624 to (527.04, 545.44, 24) mm, rotated rx -180 ry 0 rz 160 deg; joints [11.21, 80.938, -22.821, -144.492, 63.144, 162.134]
  Set speed (17.5 mm/s)
  Call Extruder(229.90874)
  MoveL 1625 to (526.1, 545.99, 24) mm, rotated rx 180 ry 0 rz 160 deg; joints [11.295, 80.788, -22.49, -144.455, 63.318, 162.212]
  Set speed (17.5 mm/s)
  Call Extruder(233.43502)
  MoveL 1626 to (525.14, 546.52, 24) mm, rotated rx -180 ry 0 rz 160 deg; joints [11.379, 80.635, -22.15, -144.42, 63.496, 162.294]
  Set speed (17.5 mm/s)
  Call Extruder(236.91872)
  MoveL 1627 to (524.19, 547.02, 24) mm, rotated rx 180 ry 0 rz 160 deg; joints [11.46, 80.484, -21.812, -144.387, 63.672, 162.376]
  Set speed (17.5 mm/s)
  Call Extruder(240.59405)
  MoveL 1628 to (523.17, 547.53, 24) mm, rotated rx -180 ry 0 rz 160 deg; joints [11.543, 80.322, -21.451, -144.356, 63.858, 162.466]
  Set speed (17.5 mm/s)
  Call Extruder(243.85383)
  MoveL 1629 to (522.26, 547.97, 24) mm, rotated rx -180 ry 0 rz 160 deg; joints [11.615, 80.178, -21.129, -144.33, 64.025, 162.548]
  Set speed (17.5 mm/s)
  Call Extruder(247.45319)
  MoveL 1630 to (521.24, 548.42, 24) mm, rotated rx 180 ry 0 rz 160 deg; joints [11.693, 80.017, -20.77, -144.304, 64.209, 162.641]
  Set speed (17.5 mm/s)
  Call Extruder(250.85539)
  MoveL 1631 to (520.27, 548.84, 24) mm, rotated rx -180 ry 0 rz 160 deg; joints [11.765, 79.865, -20.429, -144.28, 64.384, 162.73]
  Set speed (17.5 mm/s)
  Call Extruder(254.55899)
  MoveL 1632 to (519.21, 549.26, 24) mm, rotated rx -180 ry 0 rz 160 deg; joints [11.841, 79.698, -20.054, -144.258, 64.576, 162.83]
  Set speed (17.5 mm/s)
  Call Extruder(257.74508)
  MoveL 1633 to (518.28, 549.62, 24) mm, rotated rx -180 ry 0 rz 160 deg; joints [11.905, 79.554, -19.731, -144.24, 64.74, 162.917]
  Set speed (17.5 mm/s)
  Call Extruder(260.95510)
  MoveL 1634 to (517.35, 549.95, 24) mm, rotated rx 180 ry 0 rz 160 deg; joints [11.967, 79.408, -19.402, -144.224, 64.907, 163.007]
  Call Extruder(265.04379)
  MoveL 1635 to (516.15, 550.36, 24) mm, rotated rx -180 ry 0 rz 160 deg; joints [12.045, 79.222, -18.981, -144.206, 65.119, 163.124]
  Set speed (17.5 mm/s)
  Call Extruder(268.40453)
  MoveL 1636 to (515.15, 550.66, 24) mm, rotated rx -180 ry 0 rz 160 deg; joints [12.106, 79.067, -18.633, -144.195, 65.295, 163.222]
  Set speed (17.5 mm/s)
  Call Extruder(271.94145)
  MoveL 1637 to (514.1, 550.97, 24) mm, rotated rx 180 ry 0 rz 160 deg; joints [12.169, 78.905, -18.265, -144.183, 65.479, 163.326]
  Set speed (17.5 mm/s)
  Call Extruder(278.72537)
  MoveL 1638 to (512.06, 551.49, 24) mm, rotated rx 180 ry 0 rz 160 deg; joints [12.283, 78.593, -17.555, -144.169, 65.834, 163.533]
  Set speed (17.5 mm/s)
  Call Extruder(285.84599)
  MoveL 1639 to (509.9, 551.95, 24) mm, rotated rx -180 ry 0 rz 160 deg; joints [12.393, 78.263, -16.804, -144.162, 66.207, 163.755]
  Set speed (17.5 mm/s)
  Call Extruder(293.06078)
  MoveL 1640 to (507.7, 552.32, 24) mm, rotated rx 180 ry 0 rz 160 deg; joints [12.496, 77.929, -16.039, -144.165, 66.585, 163.988]
  Set speed (17.5 mm/s)
  Call Extruder(299.69039)
  MoveL 1641 to (505.66, 552.58, 24) mm, rotated rx -180 ry 0 rz 160 deg; joints [12.581, 77.622, -15.334, -144.176, 66.931, 164.206]
  Set speed (17.5 mm/s)
  Call Extruder(306.80180)
  MoveL 1642 to (503.46, 552.77, 24) mm, rotated rx 180 ry 0 rz 160 deg; joints [12.663, 77.293, -14.575, -144.197, 67.302, 164.446]
  Set speed (17.5 mm/s)
  Call Extruder(313.83135)
  MoveL 1643 to (501.28, 552.87, 24) mm, rotated rx -180 ry 0 rz 160 deg; joints [12.734, 76.97, -13.825, -144.225, 67.666, 164.687]
  Call Extruder(320.62464)
  MoveL 1644 to (499.17, 552.87, 24) mm, rotated rx 180 ry 0 rz 160 deg; joints [12.793, 76.659, -13.102, -144.262, 68.017, 164.925]
  Set speed (10.0 mm/s)
  MoveL 1645 to (499.17, 552.87, 28) mm, rotated rx -180 ry 0 rz 160 deg; joints [12.793, 75.932, -12.569, -144.216, 67.859, 164.802]
  Set speed (120.0 mm/s)
  MoveL 1646 to (499.13, 553.83, 28) mm, rotated rx 180 ry 0 rz 160 deg; joints [12.911, 75.958, -12.629, -144.086, 67.862, 164.734]
  Set speed (17.5 mm/s)
  Call Extruder(327.78303)
  MoveL 1647 to (496.91, 553.75, 28) mm, rotated rx 180 ry 0 rz 160 deg; joints [12.963, 75.632, -11.87, -144.134, 68.226, 164.988]
  Set speed (17.5 mm/s)
  Call Extruder(334.90097)
  MoveL 1648 to (494.71, 553.58, 28) mm, rotated rx -180 ry 0 rz 160 deg; joints [13.004, 75.311, -11.12, -144.191, 68.585, 165.242]
  Set speed (17.5 mm/s)
  Call Extruder(341.94029)
  MoveL 1649 to (492.54, 553.32, 28) mm, rotated rx 180 ry 0 rz 160 deg; joints [13.034, 74.996, -10.381, -144.256, 68.937, 165.497]
  Call Extruder(349.00522)
  MoveL 1650 to (490.38, 552.97, 28) mm, rotated rx -180 ry 0 rz 160 deg; joints [13.052, 74.684, -9.645, -144.331, 69.286, 165.755]
  Set speed (17.5 mm/s)
  Call Extruder(356.22095)
  MoveL 1651 to (488.18, 552.53, 28) mm, rotated rx -180 ry 0 rz 160 deg; joints [13.061, 74.369, -8.9, -144.417, 69.638, 166.02]
  Set speed (17.5 mm/s)
  Call Extruder(363.10119)
  MoveL 1652 to (486.11, 552.02, 28) mm, rotated rx 180 ry 0 rz 160 deg; joints [13.057, 74.074, -8.196, -144.508, 69.969, 166.274]
  Set speed (17.5 mm/s)
  Call Extruder(370.40580)
  MoveL 1653 to (483.93, 551.39, 28) mm, rotated rx 180 ry 0 rz 160 deg; joints [13.041, 73.765, -7.457, -144.614, 70.316, 166.545]
  Set speed (17.5 mm/s)
  Call Extruder(377.32389)
  MoveL 1654 to (481.9, 550.7, 28) mm, rotated rx 180 ry 0 rz 160 deg; joints [13.015, 73.477, -6.765, -144.724, 70.639, 166.802]
  Set speed (17.5 mm/s)
  Call Extruder(384.38410)
  MoveL 1655 to (479.85, 549.92, 28) mm, rotated rx 180 ry 0 rz 160 deg; joints [12.976, 73.189, -6.07, -144.846, 70.963, 167.064]
  Set speed (17.5 mm/s)
  Call Extruder(388.09926)
  MoveL 1656 to (478.79, 549.48, 28) mm, rotated rx 180 ry 0 rz 160 deg; joints [12.95, 73.04, -5.708, -144.914, 71.131, 167.201]
  Call Extruder(391.42728)
  MoveL 1657 to (477.84, 549.07, 28) mm, rotated rx -180 ry 0 rz 160 deg; joints [12.925, 72.908, -5.387, -144.977, 71.28, 167.324]
  Set speed (17.5 mm/s)
  Call Extruder(395.13816)
  MoveL 1658 to (476.8, 548.58, 28) mm, rotated rx 180 ry 0 rz 160 deg; joints [12.894, 72.762, -5.032, -145.05, 71.445, 167.461]
  Set speed (17.5 mm/s)
  Call Extruder(400.38932)
  MoveL 1659 to (475.34, 547.86, 28) mm, rotated rx 180 ry 0 rz 160 deg; joints [12.845, 72.558, -4.535, -145.156, 71.675, 167.654]
  Set speed (17.5 mm/s)
  Call Extruder(406.53010)
  MoveL 1660 to (473.66, 546.96, 28) mm, rotated rx 180 ry 0 rz 160 deg; joints [12.777, 72.326, -3.964, -145.29, 71.939, 167.879]
  Set speed (17.5 mm/s)
  Call Extruder(409.42557)
  MoveL 1661 to (472.88, 546.51, 28) mm, rotated rx -180 ry 0 rz 160 deg; joints [12.743, 72.217, -3.697, -145.354, 72.062, 167.985]
  Set speed (17.5 mm/s)
  Call Extruder(412.88082)
  MoveL 1662 to (471.96, 545.96, 28) mm, rotated rx 180 ry 0 rz 160 deg; joints [12.698, 72.09, -3.382, -145.434, 72.207, 168.111]
  Set speed (17.5 mm/s)
  Call Extruder(416.43265)
  MoveL 1663 to (471.02, 545.38, 28) mm, rotated rx -180 ry 0 rz 160 deg; joints [12.65, 71.96, -3.062, -145.518, 72.354, 168.239]
  Set speed (17.5 mm/s)
  Call Extruder(419.91011)
  MoveL 1664 to (470.12, 544.79, 28) mm, rotated rx -180 ry 0 rz 160 deg; joints [12.599, 71.835, -2.752, -145.603, 72.496, 168.364]
  Set speed (17.5 mm/s)
  Call Extruder(423.53997)
  MoveL 1665 to (469.19, 544.15, 28) mm, rotated rx -180 ry 0 rz 160 deg; joints [12.544, 71.707, -2.433, -145.694, 72.642, 168.494]
  Set speed (17.5 mm/s)
  Call Extruder(427.02423)
  MoveL 1666 to (468.31, 543.52, 28) mm, rotated rx 180 ry 0 rz 160 deg; joints [12.487, 71.585, -2.13, -145.784, 72.781, 168.618]
  Call Extruder(430.61585)
  MoveL 1667 to (467.41, 542.86, 28) mm, rotated rx -180 ry 0 rz 160 deg; joints [12.426, 71.462, -1.823, -145.879, 72.922, 168.745]
  Set speed (17.5 mm/s)
  Call Extruder(434.11513)
  MoveL 1668 to (466.56, 542.19, 28) mm, rotated rx 180 ry 0 rz 160 deg; joints [12.363, 71.344, -1.527, -145.973, 73.056, 168.868]
  Set speed (17.5 mm/s)
  Call Extruder(438.30999)
  MoveL 1669 to (465.55, 541.37, 28) mm, rotated rx 180 ry 0 rz 160 deg; joints [12.284, 71.205, -1.178, -146.09, 73.215, 169.014]
  Set speed (17.5 mm/s)
  Call Extruder(441.26028)
  MoveL 1670 to (464.85, 540.78, 28) mm, rotated rx 180 ry 0 rz 160 deg; joints [12.226, 71.108, -0.936, -146.174, 73.325, 169.116]
  Call Extruder(444.88098)
  MoveL 1671 to (464, 540.04, 28) mm, rotated rx -180 ry 0 rz 160 deg; joints [12.152, 70.992, -0.643, -146.279, 73.458, 169.24]
  Set speed (17.5 mm/s)
  Call Extruder(448.32876)
  MoveL 1672 to (463.22, 539.32, 28) mm, rotated rx 180 ry 0 rz 160 deg; joints [12.079, 70.884, -0.369, -146.382, 73.583, 169.358]
  Set speed (17.5 mm/s)
  Call Extruder(451.99722)
  MoveL 1673 to (462.39, 538.53, 28) mm, rotated rx 180 ry 0 rz 160 deg; joints [11.998, 70.77, -0.082, -146.493, 73.712, 169.481]
  Set speed (17.5 mm/s)
  Call Extruder(455.43252)
  MoveL 1674 to (461.64, 537.78, 28) mm, rotated rx 180 ry 0 rz 160 deg; joints [11.919, 70.666, 0.183, -146.599, 73.832, 169.596]
  Set speed (17.5 mm/s)
  Call Extruder(458.99439)
  MoveL 1675 to (460.87, 536.98, 28) mm, rotated rx 180 ry 0 rz 160 deg; joints [11.834, 70.56, 0.452, -146.712, 73.953, 169.713]
  Set speed (17.5 mm/s)
  Call Extruder(465.28457)
  MoveL 1676 to (459.56, 535.54, 28) mm, rotated rx -180 ry 0 rz 160 deg; joints [11.677, 70.379, 0.915, -146.917, 74.161, 169.918]
  Call Extruder(469.64640)
  MoveL 1677 to (458.68, 534.51, 28) mm, rotated rx -180 ry 0 rz 160 deg; joints [11.564, 70.257, 1.227, -147.062, 74.301, 170.057]
  Set speed (17.5 mm/s)
  Call Extruder(473.20337)
  MoveL 1678 to (457.98, 533.66, 28) mm, rotated rx 180 ry 0 rz 160 deg; joints [11.467, 70.161, 1.475, -147.184, 74.412, 170.169]
  Set speed (17.5 mm/s)
  Call Extruder(476.76870)
  MoveL 1679 to (457.3, 532.79, 28) mm, rotated rx -180 ry 0 rz 160 deg; joints [11.368, 70.066, 1.72, -147.308, 74.521, 170.28]
  Set speed (17.5 mm/s)
  Call Extruder(480.30157)
  MoveL 1680 to (456.64, 531.91, 28) mm, rotated rx -180 ry 0 rz 160 deg; joints [11.267, 69.974, 1.956, -147.433, 74.626, 170.389]
  Call Extruder(483.85897)
  MoveL 1681 to (455.99, 531.01, 28) mm, rotated rx -180 ry 0 rz 160 deg; joints [11.163, 69.884, 2.189, -147.56, 74.729, 170.496]
  Call Extruder(487.39662)
  MoveL 1682 to (455.37, 530.11, 28) mm, rotated rx -180 ry 0 rz 160 deg; joints [11.056, 69.797, 2.415, -147.689, 74.828, 170.602]
  Call Extruder(490.95980)
  MoveL 1683 to (454.76, 529.19, 28) mm, rotated rx -180 ry 0 rz 160 deg; joints [10.946, 69.712, 2.637, -147.821, 74.926, 170.707]
  Set speed (17.5 mm/s)
  Call Extruder(494.42804)
  MoveL 1684 to (454.19, 528.28, 28) mm, rotated rx 180 ry 0 rz 160 deg; joints [10.837, 69.631, 2.847, -147.952, 75.018, 170.807]
  Set speed (17.5 mm/s)
  Call Extruder(498.05182)
  MoveL 1685 to (453.61, 527.32, 28) mm, rotated rx -180 ry 0 rz 160 deg; joints [10.72, 69.549, 3.061, -148.09, 75.112, 170.91]
  Call Extruder(501.60548)
  MoveL 1686 to (453.06, 526.36, 28) mm, rotated rx 180 ry 0 rz 160 deg; joints [10.603, 69.47, 3.265, -148.227, 75.2, 171.01]
  Set speed (17.5 mm/s)
  Call Extruder(505.08645)
  MoveL 1687 to (452.54, 525.41, 28) mm, rotated rx 180 ry 0 rz 160 deg; joints [10.486, 69.396, 3.459, -148.363, 75.284, 171.105]
  Set speed (17.5 mm/s)
  Call Extruder(508.68320)
  MoveL 1688 to (452.02, 524.42, 28) mm, rotated rx -180 ry 0 rz 160 deg; joints [10.362, 69.322, 3.654, -148.506, 75.368, 171.202]
  Set speed (17.5 mm/s)
  Call Extruder(512.34560)
  MoveL 1689 to (451.51, 523.41, 28) mm, rotated rx -180 ry 0 rz 160 deg; joints [10.234, 69.249, 3.846, -148.653, 75.45, 171.299]
  Set speed (17.5 mm/s)
  Call Extruder(519.34724)
  MoveL 1690 to (450.61, 521.43, 28) mm, rotated rx 180 ry 0 rz 160 deg; joints [9.983, 69.117, 4.195, -148.939, 75.597, 171.479]
  Call Extruder(526.31332)
  MoveL 1691 to (449.79, 519.43, 28) mm, rotated rx 180 ry 0 rz 160 deg; joints [9.724, 68.995, 4.518, -149.229, 75.732, 171.651]
  Set speed (17.5 mm/s)
  Call Extruder(529.56602)
  MoveL 1692 to (449.44, 518.49, 28) mm, rotated rx 180 ry 0 rz 160 deg; joints [9.601, 68.941, 4.66, -149.366, 75.79, 171.729]
  Call Extruder(533.73229)
  MoveL 1693 to (449.01, 517.27, 28) mm, rotated rx -180 ry 0 rz 160 deg; joints [9.441, 68.875, 4.835, -149.544, 75.861, 171.826]
  Set speed (17.5 mm/s)
  Call Extruder(540.53429)
  MoveL 1694 to (448.37, 515.26, 28) mm, rotated rx 180 ry 0 rz 160 deg; joints [9.173, 68.775, 5.101, -149.838, 75.967, 171.979]
  Set speed (17.5 mm/s)
  Call Extruder(544.29057)
  MoveL 1695 to (448.06, 514.14, 28) mm, rotated rx -180 ry 0 rz 160 deg; joints [9.023, 68.725, 5.236, -150.002, 76.019, 172.06]
  Call Extruder(547.93390)
  MoveL 1696 to (447.76, 513.05, 28) mm, rotated rx -180 ry 0 rz 160 deg; joints [8.876, 68.677, 5.363, -150.162, 76.068, 172.137]
  Call Extruder(551.36983)
  MoveL 1697 to (447.52, 512.01, 28) mm, rotated rx -180 ry 0 rz 160 deg; joints [8.735, 68.636, 5.474, -150.314, 76.108, 172.207]
  Call Extruder(554.71422)
  MoveL 1698 to (447.3, 511, 28) mm, rotated rx -180 ry 0 rz 160 deg; joints [8.597, 68.597, 5.577, -150.463, 76.146, 172.274]
  Set speed (17.5 mm/s)
  Call Extruder(562.06817)
  MoveL 1699 to (446.88, 508.76, 28) mm, rotated rx 180 ry 0 rz 160 deg; joints [8.288, 68.52, 5.783, -150.793, 76.218, 172.414]
  Set speed (17.5 mm/s)
  Call Extruder(569.15882)
  MoveL 1700 to (446.56, 506.58, 28) mm, rotated rx 180 ry 0 rz 160 deg; joints [7.986, 68.457, 5.954, -151.115, 76.272, 172.541]
  Call Extruder(576.25512)
  MoveL 1701 to (446.34, 504.39, 28) mm, rotated rx 180 ry 0 rz 160 deg; joints [7.679, 68.403, 6.097, -151.438, 76.311, 172.66]
  Set speed (17.5 mm/s)
  Call Extruder(583.20951)
  MoveL 1702 to (446.21, 502.24, 28) mm, rotated rx 180 ry 0 rz 160 deg; joints [7.375, 68.361, 6.211, -151.757, 76.336, 172.768]
  Call Extruder(590.37197)
  MoveL 1703 to (446.16, 500.01, 28) mm, rotated rx 180 ry 0 rz 160 deg; joints [7.059, 68.328, 6.3, -152.086, 76.346, 172.872]
  Set speed (17.5 mm/s)
  Call Extruder(596.83881)
  MoveL 1704 to (446.2, 498.01, 28) mm, rotated rx 180 ry 0 rz 160 deg; joints [6.772, 68.307, 6.357, -152.383, 76.342, 172.958]
  Set speed (17.5 mm/s)
  Call Extruder(603.15188)
  MoveL 1705 to (446.31, 496.05, 28) mm, rotated rx -180 ry 0 rz 160 deg; joints [6.491, 68.295, 6.39, -152.673, 76.326, 173.036]
  Set speed (17.5 mm/s)
  Call Extruder(609.73545)
  MoveL 1706 to (446.49, 494.02, 28) mm, rotated rx -180 ry 0 rz 160 deg; joints [6.197, 68.291, 6.4, -152.974, 76.296, 173.11]
  Set speed (17.5 mm/s)
  Call Extruder(615.83486)
  MoveL 1707 to (446.74, 492.14, 28) mm, rotated rx 180 ry 0 rz 160 deg; joints [5.925, 68.296, 6.387, -153.252, 76.257, 173.172]
  Set speed (17.5 mm/s)
  Call Extruder(622.38758)
  MoveL 1708 to (447.07, 490.14, 28) mm, rotated rx -180 ry 0 rz 160 deg; joints [5.633, 68.309, 6.351, -153.547, 76.202, 173.233]
  Set speed (17.5 mm/s)
  Call Extruder(628.63053)
  MoveL 1709 to (447.46, 488.24, 28) mm, rotated rx -180 ry 0 rz 160 deg; joints [5.356, 68.33, 6.295, -153.827, 76.138, 173.284]
  Set speed (17.5 mm/s)
  Call Extruder(635.08937)
  MoveL 1710 to (447.94, 486.29, 28) mm, rotated rx -180 ry 0 rz 160 deg; joints [5.071, 68.36, 6.214, -154.113, 76.058, 173.331]
  Set speed (17.5 mm/s)
  Call Extruder(641.36869)
  MoveL 1711 to (448.47, 484.41, 28) mm, rotated rx 180 ry 0 rz 160 deg; joints [4.796, 68.398, 6.113, -154.387, 75.969, 173.371]
  Set speed (17.5 mm/s)
  Call Extruder(647.85085)
  MoveL 1712 to (449.09, 482.5, 28) mm, rotated rx -180 ry 0 rz 160 deg; joints [4.515, 68.445, 5.986, -154.666, 75.865, 173.405]
  Call Extruder(654.17011)
  MoveL 1713 to (449.76, 480.66, 28) mm, rotated rx 180 ry 0 rz 160 deg; joints [4.244, 68.499, 5.84, -154.934, 75.751, 173.433]
  Set speed (17.5 mm/s)
  Call Extruder(659.82470)
  MoveL 1714 to (450.41, 479.03, 28) mm, rotated rx 180 ry 0 rz 160 deg; joints [4.006, 68.554, 5.692, -155.169, 75.64, 173.453]
  Set speed (17.5 mm/s)
  Call Extruder(667.24229)
  MoveL 1715 to (451.35, 476.93, 28) mm, rotated rx 180 ry 0 rz 160 deg; joints [3.697, 68.637, 5.471, -155.47, 75.478, 173.472]
  Set speed (17.5 mm/s)
  Call Extruder(673.50238)
  MoveL 1716 to (452.22, 475.19, 28) mm, rotated rx -180 ry 0 rz 160 deg; joints [3.442, 68.715, 5.261, -155.718, 75.33, 173.482]
  Set speed (17.5 mm/s)
  Call Extruder(679.80148)
  MoveL 1717 to (453.15, 473.48, 28) mm, rotated rx -180 ry 0 rz 160 deg; joints [3.19, 68.802, 5.03, -155.961, 75.169, 173.487]
  Set speed (17.5 mm/s)
  Call Extruder(686.27956)
  MoveL 1718 to (454.17, 471.74, 28) mm, rotated rx 180 ry 0 rz 160 deg; joints [2.937, 68.899, 4.771, -156.204, 74.993, 173.486]
  Set speed (17.5 mm/s)
  Call Extruder(692.57292)
  MoveL 1719 to (455.23, 470.1, 28) mm, rotated rx -180 ry 0 rz 160 deg; joints [2.697, 69.002, 4.499, -156.432, 74.811, 173.48]
  Set speed (17.5 mm/s)
  Call Extruder(698.88500)
  MoveL 1720 to (456.35, 468.49, 28) mm, rotated rx 180 ry 0 rz 160 deg; joints [2.463, 69.113, 4.205, -156.654, 74.617, 173.468]
  Call Extruder(705.43907)
  MoveL 1721 to (457.57, 466.86, 28) mm, rotated rx 180 ry 0 rz 160 deg; joints [2.227, 69.236, 3.881, -156.875, 74.405, 173.451]
  Set speed (17.5 mm/s)
  Call Extruder(711.72757)
  MoveL 1722 to (458.8, 465.35, 28) mm, rotated rx -180 ry 0 rz 160 deg; joints [2.008, 69.362, 3.549, -157.079, 74.19, 173.428]
  Call Extruder(718.15349)
  MoveL 1723 to (460.11, 463.85, 28) mm, rotated rx 180 ry 0 rz 160 deg; joints [1.791, 69.499, 3.191, -157.278, 73.961, 173.4]
  Set speed (17.5 mm/s)
  Call Extruder(724.58758)
  MoveL 1724 to (461.48, 462.39, 28) mm, rotated rx 180 ry 0 rz 160 deg; joints [1.583, 69.644, 2.813, -157.468, 73.722, 173.367]
  Set speed (17.5 mm/s)
  Call Extruder(730.88786)
  MoveL 1725 to (462.87, 461.02, 28) mm, rotated rx -180 ry 0 rz 160 deg; joints [1.387, 69.793, 2.425, -157.644, 73.479, 173.329]
  Set speed (17.5 mm/s)
  Call Extruder(737.32683)
  MoveL 1726 to (464.34, 459.67, 28) mm, rotated rx 180 ry 0 rz 160 deg; joints [1.194, 69.953, 2.01, -157.814, 73.221, 173.286]
  Call Extruder(743.70680)
  MoveL 1727 to (465.84, 458.38, 28) mm, rotated rx 180 ry 0 rz 160 deg; joints [1.013, 70.119, 1.581, -157.973, 72.956, 173.237]
  Set speed (17.5 mm/s)
  Call Extruder(750.42207)
  MoveL 1728 to (467.48, 457.09, 28) mm, rotated rx 180 ry 0 rz 160 deg; joints [0.832, 70.302, 1.112, -158.128, 72.669, 173.181]
  Set speed (17.5 mm/s)
  Call Extruder(755.89494)
  MoveL 1729 to (468.85, 456.09, 28) mm, rotated rx 180 ry 0 rz 160 deg; joints [0.691, 70.457, 0.716, -158.246, 72.429, 173.131]
  Set speed (17.5 mm/s)
  Call Extruder(762.72738)
  MoveL 1730 to (470.6, 454.9, 28) mm, rotated rx 180 ry 0 rz 160 deg; joints [0.526, 70.657, 0.205, -158.381, 72.12, 173.063]
  Set speed (17.5 mm/s)
  Call Extruder(769.31629)
  MoveL 1731 to (472.33, 453.82, 28) mm, rotated rx -180 ry 0 rz 160 deg; joints [0.377, 70.859, -0.305, -158.5, 71.815, 172.991]
  Set speed (17.5 mm/s)
